ACTION A_Test_Motion:
T_Delay_RB_A_Tool_1 (PT:=T#500MS);
T_Delay_RB_A_Tool_2 (PT:=T#500MS);
IF A_Test_Motion_Run THEN
	CASE Process_A_Test OF
		0: // Point 0
			M_CHOOSE_POS(DATA := Move_Point_Para_A.Hand_Type, ID := 0, XYR_CONST := TRUE, Z_CONST:= FALSE);
			IF NOT Move_Point_Para_A.Enable THEN
				Move_Point_Para_A.Enable := TRUE;
				Move_Point_Para_A.Move_Type := 0;
			END_IF
			IF Move_RB_A.Done AND NOT Move_RB_A.Busy THEN	
				Process_A_Test := Process_A_Test + 5;
				Move_Point_Para_A.Enable := FALSE;
			END_IF;
		5: // Point 1
			M_CHOOSE_POS(DATA := Move_Point_Para_A.Hand_Type, ID := 0, XYR_CONST := FALSE, Z_CONST:= FALSE);
			IF NOT Move_Point_Para_A.Enable THEN
				Move_Point_Para_A.Enable := TRUE;
				Move_Point_Para_A.Move_Type := 0;
			END_IF
			IF Move_RB_A.Done AND NOT Move_RB_A.Busy THEN	
				Process_A_Test := Process_A_Test + 5;
				Move_Point_Para_A.Enable := FALSE;
			END_IF;
		10: // Point 2 - BF Pick T1 - 1
			M_CHOOSE_POS(DATA := Move_Point_Para_A.Hand_Type, ID := 1, XYR_CONST := FALSE, Z_CONST:= FALSE);
			IF NOT Move_Point_Para_A.Enable THEN
				Move_Point_Para_A.Enable := TRUE;
				Move_Point_Para_A.Move_Type := 0;
			END_IF
			IF Move_RB_A.Done AND NOT Move_RB_A.Busy THEN	
				Process_A_Test := Process_A_Test + 10;
				Move_Point_Para_A.Enable := FALSE;
			END_IF;
		20: // Point 3 - Pick Product by Tool 1 - 1
			M_CHOOSE_POS(DATA := Move_Point_Para_A.Hand_Type, ID := 2, XYR_CONST := FALSE, Z_CONST:= FALSE);
			IF NOT Move_Point_Para_A.Enable THEN
				Move_Point_Para_A.Enable := TRUE;
				Move_Point_Para_A.Move_Type := 0;
			END_IF
			IF Move_RB_A.Done AND NOT Move_RB_A.Busy THEN	
				GVL.RB_A_.Tool_1 := 1;
				T_Delay_RB_A_Tool_1.IN := TRUE;
				
			END_IF;
			IF T_Delay_RB_A_Tool_1.Q THEN	
				Move_Point_Para_A.Enable := FALSE;
				T_Delay_RB_A_Tool_1.IN := FALSE;
				Process_A_Test := Process_A_Test + 10;
			END_IF;
		30: // Point 2 - Return BF Pick T1 -1
			M_CHOOSE_POS(DATA := Move_Point_Para_A.Hand_Type, ID := 1, XYR_CONST := FALSE, Z_CONST:= FALSE);
			IF NOT Move_Point_Para_A.Enable THEN
				Move_Point_Para_A.Enable := TRUE;
				Move_Point_Para_A.Move_Type := 0;
			END_IF
			IF Move_RB_A.Done AND NOT Move_RB_A.Busy THEN	
				Process_A_Test := Process_A_Test + 10;
				Move_Point_Para_A.Enable := FALSE;
			END_IF;
				
		40: // Point 4 - BF Place T1 - 1
			M_CHOOSE_POS(DATA := Move_Point_Para_A.Hand_Type, ID := 3, XYR_CONST := FALSE, Z_CONST:= FALSE);
			IF NOT Move_Point_Para_A.Enable THEN
				Move_Point_Para_A.Enable := TRUE;
				Move_Point_Para_A.Move_Type := 0;
			END_IF
			IF Move_RB_A.Done AND NOT Move_RB_A.Busy THEN	
				Process_A_Test := Process_A_Test + 10;
				Move_Point_Para_A.Enable := FALSE;
			END_IF;
		
		50: // Point 5 - Place T1 - 1 
			M_CHOOSE_POS(DATA := Move_Point_Para_A.Hand_Type, ID := 4, XYR_CONST := FALSE, Z_CONST:= FALSE);
			IF NOT Move_Point_Para_A.Enable THEN
				Move_Point_Para_A.Enable := TRUE;
				Move_Point_Para_A.Move_Type := 0;
			END_IF
			IF Move_RB_A.Done AND NOT Move_RB_A.Busy THEN	
				GVL.RB_A_.Tool_1 := 0;
				T_Delay_RB_A_Tool_1.IN := TRUE;
				//Move_Point_Para_A.Enable := FALSE;
			END_IF;
			
			IF T_Delay_RB_A_Tool_1.Q THEN			
				Move_Point_Para_A.Enable := FALSE;
				T_Delay_RB_A_Tool_1.IN := FALSE;
				Process_A_Test := Process_A_Test + 10;
			END_IF
		
		60: // Point 4 - BF Place T1 - 1
			M_CHOOSE_POS(DATA := Move_Point_Para_A.Hand_Type, ID := 3, XYR_CONST := FALSE, Z_CONST:= FALSE);
			IF NOT Move_Point_Para_A.Enable THEN
				Move_Point_Para_A.Enable := TRUE;
				Move_Point_Para_A.Move_Type := 0;
			END_IF
			IF Move_RB_A.Done AND NOT Move_RB_A.Busy THEN	
				Process_A_Test := Process_A_Test + 10;
				Move_Point_Para_A.Enable := FALSE;
			END_IF;
			
		70: // Point 6 - BF Pick T1-2
			M_CHOOSE_POS(DATA := Move_Point_Para_A.Hand_Type, ID := 5, XYR_CONST := FALSE, Z_CONST:= FALSE);
			IF NOT Move_Point_Para_A.Enable THEN
				Move_Point_Para_A.Enable := TRUE;
				Move_Point_Para_A.Move_Type := 0;
			END_IF
			IF Move_RB_A.Done AND NOT Move_RB_A.Busy THEN	
				Process_A_Test := Process_A_Test + 10;
				Move_Point_Para_A.Enable := FALSE;
			END_IF;
		80: // Point 7 - Pick Tool 1 - 2
			M_CHOOSE_POS(DATA := Move_Point_Para_A.Hand_Type, ID := 6, XYR_CONST := FALSE, Z_CONST:= FALSE);
			IF NOT Move_Point_Para_A.Enable THEN
				Move_Point_Para_A.Enable := TRUE;
				Move_Point_Para_A.Move_Type := 0;
			END_IF
			IF Move_RB_A.Done AND NOT Move_RB_A.Busy THEN	
				GVL.RB_A_.Tool_1 := 1;
				T_Delay_RB_A_Tool_2.IN := TRUE;
				//Move_Point_Para_A.Enable := FALSE;
			END_IF;
			IF T_Delay_RB_A_Tool_2.Q THEN
				T_Delay_RB_A_Tool_2.IN := FALSE;
				Move_Point_Para_A.Enable := FALSE;
				Process_A_Test := Process_A_Test + 10;
			END_IF;
		90: // Point 6 - Return BF Pick T1 - 2 
			M_CHOOSE_POS(DATA := Move_Point_Para_A.Hand_Type, ID := 5, XYR_CONST := FALSE, Z_CONST:= FALSE);
			IF NOT Move_Point_Para_A.Enable THEN
				Move_Point_Para_A.Enable := TRUE;
				Move_Point_Para_A.Move_Type := 0;
			END_IF
			IF Move_RB_A.Done AND NOT Move_RB_A.Busy THEN	
				Process_A_Test := Process_A_Test + 10;
				Move_Point_Para_A.Enable := FALSE;
			END_IF;
				
		100: // Point 8 - BF Place T1 - 2 
			M_CHOOSE_POS(DATA := Move_Point_Para_A.Hand_Type, ID := 7, XYR_CONST := FALSE, Z_CONST:= FALSE);
			IF NOT Move_Point_Para_A.Enable THEN
				Move_Point_Para_A.Enable := TRUE;
				Move_Point_Para_A.Move_Type := 0;
			END_IF
			IF Move_RB_A.Done AND NOT Move_RB_A.Busy THEN	
				Process_A_Test := Process_A_Test + 10;
				Move_Point_Para_A.Enable := FALSE;
			END_IF;
		
		110: // Point 9 - Place T2
			M_CHOOSE_POS(DATA := Move_Point_Para_A.Hand_Type, ID := 8, XYR_CONST := FALSE, Z_CONST:= FALSE);
			IF NOT Move_Point_Para_A.Enable THEN
				Move_Point_Para_A.Enable := TRUE;
				Move_Point_Para_A.Move_Type := 0;
			END_IF
			IF Move_RB_A.Done AND NOT Move_RB_A.Busy THEN	
				GVL.RB_A_.Tool_1 := 0;
				T_Delay_RB_A_Tool_2.IN := TRUE;
				//Move_Point_Para_A.Enable := FALSE;
			END_IF;
			
			IF T_Delay_RB_A_Tool_2.Q THEN			
				T_Delay_RB_A_Tool_2.IN := FALSE;
				Move_Point_Para_A.Enable := FALSE;
				Process_A_Test := Process_A_Test + 10;
			END_IF
		
		120: // Point 8 - BF Place T2
			M_CHOOSE_POS(DATA := Move_Point_Para_A.Hand_Type, ID := 7, XYR_CONST := FALSE, Z_CONST:= FALSE);
			IF NOT Move_Point_Para_A.Enable THEN
				Move_Point_Para_A.Enable := TRUE;
				Move_Point_Para_A.Move_Type := 0;
			END_IF
			IF Move_RB_A.Done AND NOT Move_RB_A.Busy THEN	
				Process_A_Test := Process_A_Test + 10;
				Move_Point_Para_A.Enable := FALSE;
			END_IF;
			
		
		130: // WAIT XYR
			Process_A_Test := 5;
			A_Test_Motion_Finish := TRUE;
		
	END_CASE
ELSE
	Process_A_Test := 0;
END_IF
END_ACTION

ACTION B1_Test_Motion:
Ton_Test_B(PT := T#500MS);
T_Delay_RB_B_Tool_1(PT := T#500MS);
T_Delay_RB_B_Tool_2(PT := T#500MS);
IF B_Test_Motion_Run THEN
	CASE Process_B_Test OF
		0: // Point 0
			M_CHOOSE_POS(DATA := Move_Point_Para_B.Hand_Type, ID := 0, XYR_CONST := TRUE, Z_CONST:= FALSE);
			IF NOT Move_Point_Para_B.Enable THEN
				Move_Point_Para_B.Enable := TRUE;
				Move_Point_Para_B.Move_Type := 0;
			END_IF
			IF Move_RB_B.Done AND NOT Move_RB_B.Busy THEN	
				Process_B_Test := Process_B_Test + 5;
				Move_Point_Para_B.Enable := FALSE;
			END_IF;
		5: // Point 1
			M_CHOOSE_POS(DATA := Move_Point_Para_B.Hand_Type, ID := 0, XYR_CONST := FALSE, Z_CONST:= FALSE);
			IF NOT Move_Point_Para_B.Enable THEN
				Move_Point_Para_B.Enable := TRUE;
				Move_Point_Para_B.Move_Type := 0;
			END_IF
			IF Move_RB_B.Done AND NOT Move_RB_B.Busy THEN	
				Process_B_Test := Process_B_Test + 5;
				Move_Point_Para_B.Enable := FALSE;
			END_IF;
		10: // Point 2 - BF Pick T1
			M_CHOOSE_POS(DATA := Move_Point_Para_B.Hand_Type, ID := 1, XYR_CONST := FALSE, Z_CONST:= FALSE);
			IF NOT Move_Point_Para_B.Enable THEN
				Move_Point_Para_B.Enable := TRUE;
				Move_Point_Para_B.Move_Type := 0;
			END_IF
			IF Move_RB_B.Done AND NOT Move_RB_B.Busy THEN	
				Process_B_Test := Process_B_Test + 10;
				Move_Point_Para_B.Enable := FALSE;
			END_IF;
		
		20: // WAIT Timer
			
			Ton_Test_B.IN := TRUE;
			IF Ton_Test_B.Q THEN
				Process_B_Test := 30;
				Ton_Test_B.IN := FALSE;
			END_IF
		30: // Point 3 - Pick T1
			
			M_CHOOSE_POS(DATA := Move_Point_Para_B.Hand_Type, ID := 2, XYR_CONST := FALSE, Z_CONST:= FALSE);
			IF NOT Move_Point_Para_B.Enable THEN
				Move_Point_Para_B.Enable := TRUE;
				Move_Point_Para_B.Move_Type := 0;
			END_IF
			IF Move_RB_B.Done AND NOT Move_RB_B.Busy THEN	
				GVL.RB_B_.Tool_1 := 1;
				T_Delay_RB_B_Tool_1.IN := TRUE;
				
			END_IF;
			IF T_Delay_RB_B_Tool_1.Q THEN
				Move_Point_Para_B.Enable := FALSE;
				T_Delay_RB_B_Tool_1.IN := FALSE;
				Process_B_Test := Process_B_Test + 10;		
			END_IF;
		40: // Point 2 - BF Pick T1
			M_CHOOSE_POS(DATA := Move_Point_Para_B.Hand_Type, ID := 1, XYR_CONST := FALSE, Z_CONST:= FALSE);
			IF NOT Move_Point_Para_B.Enable THEN
				Move_Point_Para_B.Enable := TRUE;
				Move_Point_Para_B.Move_Type := 0;
			END_IF
			IF Move_RB_B.Done AND NOT Move_RB_B.Busy THEN	
				Process_B_Test := Process_B_Test + 10;
				Move_Point_Para_B.Enable := FALSE;
			END_IF;
		50: // Point 4 - BF Place T1
			M_CHOOSE_POS(DATA := Move_Point_Para_B.Hand_Type, ID := 3, XYR_CONST := FALSE, Z_CONST:= FALSE);
			IF NOT Move_Point_Para_B.Enable THEN
				Move_Point_Para_B.Enable := TRUE;
				Move_Point_Para_B.Move_Type := 0;
			END_IF
			IF Move_RB_B.Done AND NOT Move_RB_B.Busy THEN	
				Process_B_Test := Process_B_Test + 10;
				Move_Point_Para_B.Enable := FALSE;
			END_IF;
		
		60: // Point 5 - Place T1
			M_CHOOSE_POS(DATA := Move_Point_Para_B.Hand_Type, ID := 4, XYR_CONST := FALSE, Z_CONST:= FALSE);
			IF NOT Move_Point_Para_B.Enable THEN
				Move_Point_Para_B.Enable := TRUE;
				Move_Point_Para_B.Move_Type := 0;
			END_IF
			IF Move_RB_B.Done AND NOT Move_RB_B.Busy THEN	
				GVL.RB_B_.Tool_1 := 0;
				T_Delay_RB_B_Tool_1.IN := TRUE;
				
			END_IF;
			IF T_Delay_RB_B_Tool_1.Q THEN
				Move_Point_Para_B.Enable := FALSE;
				T_Delay_RB_B_Tool_1.IN := FALSE;
				Process_B_Test := Process_B_Test + 10;
				
			END_IF;
			
		70: // Point 4 - BF Place T1
			M_CHOOSE_POS(DATA := Move_Point_Para_B.Hand_Type, ID := 3, XYR_CONST := FALSE, Z_CONST:= FALSE);
			IF NOT Move_Point_Para_B.Enable THEN
				Move_Point_Para_B.Enable := TRUE;
				Move_Point_Para_B.Move_Type := 0;
			END_IF
			IF Move_RB_B.Done AND NOT Move_RB_B.Busy THEN	
				Process_B_Test := Process_B_Test + 10;
				Move_Point_Para_B.Enable := FALSE;
			END_IF;
			
		80: // Point 6 - BF Pick T2
			M_CHOOSE_POS(DATA := Move_Point_Para_B.Hand_Type, ID := 5, XYR_CONST := FALSE, Z_CONST:= FALSE);
			IF NOT Move_Point_Para_B.Enable THEN
				Move_Point_Para_B.Enable := TRUE;
				Move_Point_Para_B.Move_Type := 0;
			END_IF
			IF Move_RB_B.Done AND NOT Move_RB_B.Busy THEN	
				Process_B_Test := Process_B_Test + 10;
				Move_Point_Para_B.Enable := FALSE;
			END_IF;
		

		90: // Point 7 - Pick T2
			M_CHOOSE_POS(DATA := Move_Point_Para_B.Hand_Type, ID := 6, XYR_CONST := FALSE, Z_CONST:= FALSE);
			IF NOT Move_Point_Para_B.Enable THEN
				Move_Point_Para_B.Enable := TRUE;
				Move_Point_Para_B.Move_Type := 0;
			END_IF
			IF Move_RB_B.Done AND NOT Move_RB_B.Busy THEN	
				GVL.RB_B_.Tool_1 := 1;
				T_Delay_RB_B_Tool_2.IN := TRUE;
				
			END_IF;
			IF T_Delay_RB_B_Tool_2.Q THEN
				Move_Point_Para_B.Enable := FALSE;
				T_Delay_RB_B_Tool_2.IN := FALSE;
				Process_B_Test := Process_B_Test + 10;
				
			END_IF;
		100: // Point 6 - BF Pick T2
			M_CHOOSE_POS(DATA := Move_Point_Para_B.Hand_Type, ID := 5, XYR_CONST := FALSE, Z_CONST:= FALSE);
			IF NOT Move_Point_Para_B.Enable THEN
				Move_Point_Para_B.Enable := TRUE;
				Move_Point_Para_B.Move_Type := 0;
			END_IF
			IF Move_RB_B.Done AND NOT Move_RB_B.Busy THEN	
				Process_B_Test := Process_B_Test + 10;
				Move_Point_Para_B.Enable := FALSE;
			END_IF;
		110: // Point 8 - BF Place T2
			M_CHOOSE_POS(DATA := Move_Point_Para_B.Hand_Type, ID := 7, XYR_CONST := FALSE, Z_CONST:= FALSE);
			IF NOT Move_Point_Para_B.Enable THEN
				Move_Point_Para_B.Enable := TRUE;
				Move_Point_Para_B.Move_Type := 0;
			END_IF
			IF Move_RB_B.Done AND NOT Move_RB_B.Busy THEN	
				Process_B_Test := Process_B_Test + 10;
				Move_Point_Para_B.Enable := FALSE;
			END_IF;
		
		120: // Point 9 - Place T2
			M_CHOOSE_POS(DATA := Move_Point_Para_B.Hand_Type, ID := 8, XYR_CONST := FALSE, Z_CONST:= FALSE);
			IF NOT Move_Point_Para_B.Enable THEN
				Move_Point_Para_B.Enable := TRUE;
				Move_Point_Para_B.Move_Type := 0;
			END_IF
			IF Move_RB_B.Done AND NOT Move_RB_B.Busy THEN	
				GVL.RB_B_.Tool_1 := 0;
				T_Delay_RB_B_Tool_2.IN := TRUE;
				
			END_IF;
			IF T_Delay_RB_B_Tool_2.Q THEN
				Move_Point_Para_B.Enable := FALSE;
				T_Delay_RB_B_Tool_2.IN := FALSE;
				Process_B_Test := Process_B_Test + 10;
				
			END_IF;
			
		130: // Point 8 - BF Place T2
			M_CHOOSE_POS(DATA := Move_Point_Para_B.Hand_Type, ID := 7, XYR_CONST := FALSE, Z_CONST:= FALSE);
			IF NOT Move_Point_Para_B.Enable THEN
				Move_Point_Para_B.Enable := TRUE;
				Move_Point_Para_B.Move_Type := 0;
			END_IF
			IF Move_RB_B.Done AND NOT Move_RB_B.Busy THEN	
				Process_B_Test := Process_B_Test + 10;
				Move_Point_Para_B.Enable := FALSE;
			END_IF;
			
			
		140: // Finish
			//Ton_Test_B.IN := FALSE;
			Process_B_Test := 5;
			A_Test_Motion_Finish := TRUE;
			
		
	END_CASE
ELSE
	Process_B_Test := 0;
END_IF
END_ACTION

ACTION _Main_Process_Test_VS:
// PROCESS 
IF Ena_Test THEN
	GVL.RB_A.COORD := 1;
	GVL.RB_B.COORD := 1;
	IF NOT Just_Start_Test THEN
		A_Test_Motion_Run := FALSE;
		B_Test_Motion_Run := FALSE;
		Process_B_Test := 0;
		Process_A_Test := 0;
	END_IF
	Just_Start_Test := TRUE;
	A_Test_Motion_Run := TRUE;
	A_Test_Motion_VS();
// 	B_Test_Motion_Run := TRUE;
// 	B1_Test_Motion_VS();

ELSIF NOT Ena_Test THEN

	A_Test_Motion_Run := FALSE;
	B_Test_Motion_Run := FALSE;
	Process_B_Test := 0;
	Process_A_Test := 0;
	
END_IF	 
{endregion}
END_ACTION

ACTION A_Test_Motion_VS:
Ton_Test_A(PT := T#500MS);
IF A_Test_Motion_Run THEN
	CASE Process_A_Test OF
		0: // Point 1 - Wait
			M_CHOOSE_POS(DATA := Move_Point_Para_A.Hand_Type, ID := 0, XYR_CONST := FALSE, Z_CONST:= FALSE);
			IF NOT Move_Point_Para_A.Enable THEN
				Move_Point_Para_A.Enable := TRUE;
				Move_Point_Para_A.Move_Type := 0;
			END_IF
			IF Move_RB_A.Done AND NOT Move_RB_A.Busy THEN	
				Process_A_Test := Process_A_Test + 10;
				Move_Point_Para_A.Enable := FALSE;
			END_IF;
		10: // Point 2 - BF Pick T1
			M_CHOOSE_POS(DATA := Move_Point_Para_A.Hand_Type, ID := 1, XYR_CONST := FALSE, Z_CONST:= FALSE);
			IF NOT Move_Point_Para_A.Enable THEN
				Move_Point_Para_A.Enable := TRUE;
				Move_Point_Para_A.Move_Type := 0;
			END_IF
			IF Move_RB_A.Done AND NOT Move_RB_A.Busy THEN	
				Process_A_Test := Process_A_Test + 10;
				Move_Point_Para_A.Enable := FALSE;
			END_IF;
		20: // Point 3 - Pick T1
			M_CHOOSE_POS(DATA := Move_Point_Para_A.Hand_Type, ID := 2, XYR_CONST := FALSE, Z_CONST:= FALSE);
			IF NOT Move_Point_Para_A.Enable THEN
				Move_Point_Para_A.Enable := TRUE;
				Move_Point_Para_A.Move_Type := 0;
			END_IF
			IF Move_RB_A.Done AND NOT Move_RB_A.Busy THEN	
				Process_A_Test := Process_A_Test + 10;
				Move_Point_Para_A.Enable := FALSE;
			END_IF;
		30: // Point 4 - BF Pick T1
			M_CHOOSE_POS(DATA := Move_Point_Para_A.Hand_Type, ID := 3, XYR_CONST := FALSE, Z_CONST:= FALSE);
			IF NOT Move_Point_Para_A.Enable THEN
				Move_Point_Para_A.Enable := TRUE;
				Move_Point_Para_A.Move_Type := 0;
			END_IF
			IF Move_RB_A.Done AND NOT Move_RB_A.Busy THEN	
				Process_A_Test := Process_A_Test + 10;
				Move_Point_Para_A.Enable := FALSE;
			END_IF;
				
		40: // Point 5 - Trigger VS
			M_CHOOSE_POS(DATA := Move_Point_Para_A.Hand_Type, ID := 4, XYR_CONST := FALSE, Z_CONST:= FALSE);
			IF NOT Move_Point_Para_A.Enable THEN
				Move_Point_Para_A.Enable := TRUE;
				Move_Point_Para_A.Move_Type := 0;
			END_IF
			IF Move_RB_A.Done AND NOT Move_RB_A.Busy THEN	
				Process_A_Test := Process_A_Test + 10;
				Move_Point_Para_A.Enable := FALSE;
			END_IF;
			
		50: // WAIT Timer
			
			Ton_Test_A.IN := TRUE;
			IF Ton_Test_A.Q THEN
				Process_A_Test := Process_A_Test + 10;
				Ton_Test_A.IN := FALSE;
			END_IF
			
		60: // Trigger VS
			
			IF ( NOT GVL.Data_Calib_RB[0].Run_No_Trigger) THEN
				GVL.Auto_VS_RB[0].Enable_FB_Trigger_VS := TRUE;
				GVL.Auto_VS_RB[0].Start_FB_Trigger_VS := TRUE;
			END_IF
			
			IF ((Trigger_VS_FB[0].DoneAll AND NOT Trigger_VS_FB[0].Busy) OR GVL.Data_Calib_RB[0].Run_No_Trigger ) THEN
				GVL.Auto_VS_RB[0].Enable_FB_Trigger_VS := FALSE;
				GVL.Auto_VS_RB[0].Start_FB_Trigger_VS := FALSE;
				Process_A_Test := Process_A_Test + 10;
			END_IF;	
			
		70: // WAIT XYR
			Process_A_Test := 0;
			A_Test_Motion_Finish := TRUE;
		
	END_CASE
ELSE
	Process_A_Test := 0;
END_IF
END_ACTION

ACTION B1_Test_Motion_VS:
Ton_Test_B(PT := T#500MS);
IF B_Test_Motion_Run THEN
	CASE Process_B_Test OF
		0: // Point 1 - Wait
			M_CHOOSE_POS(DATA := Move_Point_Para_B.Hand_Type, ID := 0, XYR_CONST := FALSE, Z_CONST:= FALSE);
			IF NOT Move_Point_Para_B.Enable THEN
				Move_Point_Para_B.Enable := TRUE;
				Move_Point_Para_B.Move_Type := 0;
			END_IF
			IF Move_RB_B.Done AND NOT Move_RB_B.Busy THEN	
				Process_B_Test := Process_B_Test + 10;
				Move_Point_Para_B.Enable := FALSE;
			END_IF;
		10: // Point 2 - BF Pick T1
			M_CHOOSE_POS(DATA := Move_Point_Para_B.Hand_Type, ID := 1, XYR_CONST := FALSE, Z_CONST:= FALSE);
			IF NOT Move_Point_Para_B.Enable THEN
				Move_Point_Para_B.Enable := TRUE;
				Move_Point_Para_B.Move_Type := 0;
			END_IF
			IF Move_RB_B.Done AND NOT Move_RB_B.Busy THEN	
				Process_B_Test := Process_B_Test + 10;
				Move_Point_Para_B.Enable := FALSE;
			END_IF;
		
		20: // WAIT Timer
			Process_B_Test := Process_B_Test + 10;
// 			Ton_Test_B.IN := TRUE;
// 			IF Ton_Test_B.Q THEN
// 				Process_B_Test := 30;
// 				Ton_Test_B.IN := FALSE;
// 			END_IF
		30: // Point 3 - Pick T1
			
			M_CHOOSE_POS(DATA := Move_Point_Para_B.Hand_Type, ID := 2, XYR_CONST := FALSE, Z_CONST:= FALSE);
			IF NOT Move_Point_Para_B.Enable THEN
				Move_Point_Para_B.Enable := TRUE;
				Move_Point_Para_B.Move_Type := 0;
			END_IF
			IF Move_RB_B.Done AND NOT Move_RB_B.Busy THEN	
				Process_B_Test := Process_B_Test + 10;
				Move_Point_Para_B.Enable := FALSE;
			END_IF;
		
		40: // Point 4 - BF Pick T1
			M_CHOOSE_POS(DATA := Move_Point_Para_B.Hand_Type, ID := 3, XYR_CONST := FALSE, Z_CONST:= FALSE);
			IF NOT Move_Point_Para_B.Enable THEN
				Move_Point_Para_B.Enable := TRUE;
				Move_Point_Para_B.Move_Type := 0;
			END_IF
			IF Move_RB_B.Done AND NOT Move_RB_B.Busy THEN	
				Process_B_Test := Process_B_Test + 10;
				Move_Point_Para_B.Enable := FALSE;
			END_IF;
		50: // Point 5 - Trigger VS
			M_CHOOSE_POS(DATA := Move_Point_Para_B.Hand_Type, ID := 4, XYR_CONST := FALSE, Z_CONST:= FALSE);
			IF NOT Move_Point_Para_B.Enable THEN
				Move_Point_Para_B.Enable := TRUE;
				Move_Point_Para_B.Move_Type := 0;
			END_IF
			IF Move_RB_B.Done AND NOT Move_RB_B.Busy THEN	
				Process_B_Test := Process_B_Test + 10;
				Move_Point_Para_B.Enable := FALSE;
			END_IF;
		60: // WAIT Timer
			
			Ton_Test_B.IN := TRUE;
			IF Ton_Test_B.Q THEN
				Process_B_Test := Process_B_Test + 10;
				Ton_Test_B.IN := FALSE;
			END_IF
			
		70: // Trigger VS
			IF ( NOT GVL.Data_Calib_RB[0].Run_No_Trigger) THEN
				GVL.Auto_VS_RB[0].Enable_FB_Trigger_VS := TRUE;
				GVL.Auto_VS_RB[0].Start_FB_Trigger_VS := TRUE;
			END_IF
			
			IF ((Trigger_VS_FB[0].DoneAll AND NOT Trigger_VS_FB[0].Busy) OR GVL.Data_Calib_RB[0].Run_No_Trigger ) THEN
				GVL.Auto_VS_RB[0].Enable_FB_Trigger_VS := FALSE;
				GVL.Auto_VS_RB[0].Start_FB_Trigger_VS := FALSE;
				Process_B_Test := Process_B_Test + 10;
			END_IF;
	
		80: // Finish
			//Ton_Test_B.IN := FALSE;
			Process_B_Test := 0;
			A_Test_Motion_Finish := TRUE;
			
		
	END_CASE
ELSE
	Process_B_Test := 0;
END_IF
END_ACTION

ACTION _Main_Process_4:
// Check Pos cmp

B_Allow_NextStep := NOT GVL_2.Process3.Auto_Man_B OR nextstepRtrigB.Q;
nextstepRtrigB(CLK := ( GVL_2.Process3.Auto_Man_B AND GVL_2.Process3.NextStep_B));
A_Allow_NextStep := NOT GVL_2.Process3.Auto_Man_A OR nextstepRtrigA.Q;
nextstepRtrigA(CLK := ( GVL_2.Process3.Auto_Man_A AND GVL_2.Process3.NextStep_A));
// Clear Data
IF NOT GVL.Pro4_.Process.Clear_Data THEN
	// ko làm gì
ELSE
	GVL.Pro4_.Process.DATA_MC_TS := 0;
	GVL.Pro4_.Process.DATA_MC_VS := 0;
	GVL.Pro4_.Process.DATA_TOOL_A1_IN := 0;
	GVL.Pro4_.Process.DATA_TOOL_A2_OUT := 0;
	GVL.Pro4_.Process.DATA_TOOL_B1_IN := 0;
	GVL.Pro4_.Process.DATA_TOOL_A1_IN_OLD := 0;	
END_IF



// PROCESS 
IF Ena4 THEN
// cv-ng
CNV_NG();	
// Process MC1
Pro_MC1_4_();
// Process MC2
Pro_MC2_4_();	
// trigger
B_Trigger_4();
////// process robot A
A0_Wait_4();
A1_Pick_T1_4();
A2_Place_T1_OK_4();
A3_Place_T1_NG_4();
A4_Pick_T2_4();
A5_Place_T2_OK_4();
A6_Place_T2_NG_4();
A7_Barcode_T1_4();
A8_Place_T2_NG_TS_4();
	CASE Pro_A4 OF
	0: // INIT
			
			GVL.RB_A.COORD := 1;
			RBA_BufferMode := 0; 
	 		Wait_A4_Finish			:= FALSE;
			Pick_A4_T1_Finish 		:= FALSE;
			Pick_A4_T2_Finish		:= FALSE;
			Barcode_A4_Finish		:= FALSE;
			Place_OK_A4_T1_Finish 	:= FALSE;
			Place_Ok_A4_T2_Finish 	:= FALSE;
			Place_NG_A4_T1_Finish 	:= FALSE;
			Place_NG_A4_T2_Finish 	:= FALSE;
			Place_NG_TS_A4_T2_Finish	:= FALSE;
			
	 		Wait_A4_Run				:= FALSE;
			Pick_A4_T1_Run			:= FALSE;
			Pick_A4_T2_Run			:= FALSE;
			Barcode_A4_Run			:= FALSE;
			Place_OK_A4_T1_Run	 	:= FALSE;
			Place_Ok_A4_T2_Run	 	:= FALSE;
			Place_NG_A4_T1_Run	 	:= FALSE;
			Place_NG_A4_T2_Run		:= FALSE;			
			Place_NG_TS_A4_T2_Run	:= FALSE;	
			Pro_A4_BF := 0; // namnv
			Pro_A4 := Pro_A4 + 10; 
			
	10: // CALL WAIT	
		LOG_A.Write('Robot A to Wait');	
		IF NOT Wait_A4_Run THEN
			RBA_BufferMode := 0;
			Wait_A4_Run := TRUE;
		END_IF
		IF Wait_A4_Finish AND A_Allow_NextStep THEN
			Wait_A4_Run := FALSE;
			Pro_A4_BF := 10; // namnv
			Pro_A4 := Pro_A4 + 10;
		END_IF;		
	20: // CHECK PICK OR PLACE T1
			
		 	Wait_A4_Finish			:= FALSE;
			Pick_A4_T1_Finish 		:= FALSE;
			Pick_A4_T2_Finish		:= FALSE;
			Barcode_A4_Finish		:= FALSE;
			Place_OK_A4_T1_Finish 	:= FALSE;
			Place_Ok_A4_T2_Finish 	:= FALSE;
			Place_NG_A4_T1_Finish 	:= FALSE;
			Place_NG_A4_T2_Finish 	:= FALSE;
			Place_NG_TS_A4_T2_Finish 	:= FALSE;
			
			CASE GVL.Pro4_.Process.DATA_TOOL_A1_IN OF
				0: // none
					Pro_A4 := 30; // Pick T1
				1: // Barcode
					Pro_A4 := 40; // Barcode T1
				2: // Ok
					CASE GVL.Pro4_.Process.DATA_MC_VS OF
						2: 
							Pro_A4 := 50; // Place T1 OK => MC2
						3: 
							Pro_A4 := 25; // CHECK PICK OR PLACE T2
						4: 
							Pro_A4 := 25;
						5: 
							Pro_A4 := 25;
					END_CASE;
					
				3: // NG
					// Pro_A4 := 60;	
					// namnv NG cung van dat vao may Vision
					CASE GVL.Pro4_.Process.DATA_MC_VS OF
						2: 
							Pro_A4 := 50; // Place T1 NG => MC2
						3: 
							Pro_A4 := 25; // CHECK PICK OR PLACE T2
						4: 
							Pro_A4 := 25;
							//namnv
						5: 
							Pro_A4 := 25;	
							
					END_CASE;
					
			END_CASE
			// Pro_A4_BF := 20; // namnv
	25: // CHECK PICK OR PLACE T2
			CASE GVL.Pro4_.Process.DATA_TOOL_A2_OUT OF
				0: // none
					Pro_A4 := 70; // pick T2
				1: // have
					//Pro_B3 := 80; // Place OK CNV
				2: // OK
					Pro_A4 := 80; // Place OK CNV
				3: // NG - VS
					Pro_A4 := 90; // Place NG-VS CNV
				// namnv
				4: // NG - TS
					Pro_A4 := 100; // Place NG-TS CNV
			END_CASE	
			// Pro_A4_BF := 25; // namnv	
	30: // Pick T1
		 //DATA_MC1 := 3;
		 LOG_A.Write('Robot A Pick T1');
// 		IF NOT Pick_A4_T1_Run  AND (GVL.Pro4_.Process.DATA_MC_TS = 3 OR GVL.Pro4_.Process.DATA_MC_TS = 4) THEN
		//IF NOT Pick_B3_T1_Run THEN	
		// namnv0204
		IF NOT Pick_A4_T1_Run  AND (GVL.Pro4_.Process.DATA_MC_TS = 3 OR GVL.Pro4_.Process.DATA_MC_TS = 4 OR GVL.Pro4_.Process.DATA_MC_TS = 1) THEN
			RBA_BufferMode := 0;
			Pick_A4_T1_Run := TRUE;
		ELSIF NOT Pick_A4_T1_Run AND GVL.Pro4_.Process.DATA_MC_TS <> 3 AND GVL.Pro4_.Process.DATA_MC_TS <> 4 AND GVL.Pro4_.Process.DATA_MC_TS <> 1 THEN
			Pro_A4 := 25;
			Pro_A4_BF := 30; // namnv
		END_IF
		IF Pick_A4_T1_Finish AND A_Allow_NextStep THEN
			Pick_A4_T1_Run := FALSE;
			// Pro_A4 := 40;
			// namnv - khong cho di ra barcode luon
			Pro_A4 := 20;
			Pro_A4_BF := 30; // namnv
		END_IF;
		
	40: // Barcode T1
		LOG_A.Write('Robot A barcode T1');
		IF NOT Barcode_A4_Run THEN
			RBA_BufferMode := 0;
			Barcode_A4_Run := TRUE;
		END_IF
		IF Barcode_A4_Finish AND A_Allow_NextStep THEN
			Barcode_A4_Run := FALSE;
			// Pro_A4 := 10;
			Pro_A4 := 20;  // Khong cho chay ve wait nua  Namnv
			Pro_A4_BF := 40; // namnv
		END_IF;		
		
	50: // Place T1 OK/NG => MC2
		//DATA_MC2 := 2;
		LOG_A.Write('Robot A Place T1 OK');
		RBA_BufferMode := 1;
		IF NOT Place_OK_A4_T1_Run AND GVL.Pro4_.Process.DATA_MC_VS = 2 THEN
	
			Place_OK_A4_T1_Run := TRUE;
		END_IF
		IF Place_OK_A4_T1_Finish AND A_Allow_NextStep THEN
			Place_OK_A4_T1_Run := FALSE;
			Pro_A4 := 25;
			Pro_A4_BF := 50; // namnv
		END_IF;	
		
	60: // Place T1 NG => CNV TS NG
// 		IF NOT Place_NG_A4_T1_Run  THEN
// 			RBA_BufferMode := 1;
// 			Place_NG_A4_T1_Run := TRUE;
// 		END_IF
// 		IF Place_NG_A4_T1_Finish AND A_Allow_NextStep THEN
// 			Place_NG_A4_T1_Run := FALSE;
// 			Pro_A4 := 10;
// 			Pro_A4_BF := 60; // namnv
// 		END_IF;			
		
				
		
	70: // PICK T2
		//DATA_MC2 := 3;
		//IF NOT Pick_A4_T2_Run  AND ( GVL.Pro4_.Process.DATA_MC_VS = 3 OR GVL.Pro4_.Process.DATA_MC_VS = 4 ) THEN
		LOG_A.Write('Robot A Pick T2');
		IF NOT Pick_A4_T2_Run  AND ( GVL.Pro4_.Process.DATA_MC_VS = 3 OR GVL.Pro4_.Process.DATA_MC_VS = 4 OR GVL.Pro4_.Process.DATA_MC_VS = 5 ) THEN
			RBA_BufferMode := 1;
			Pick_A4_T2_Run := TRUE;
		ELSIF NOT Pick_A4_T2_Run AND( GVL.Pro4_.Process.DATA_MC_VS = 1 OR GVL.Pro4_.Process.DATA_MC_VS = 2) AND ( GVL.Pro4_.Process.DATA_MC_TS = 1 OR GVL.Pro4_.Process.DATA_MC_TS = 3 OR GVL.Pro4_.Process.DATA_MC_TS = 4 ) THEN
			Pro_A4 := 10;
			Pro_A4_BF := 70; // namnv
		END_IF
		IF Pick_A4_T2_Finish AND A_Allow_NextStep THEN
			Pick_A4_T2_Run := FALSE;
			Pro_A4 := 20;
			Pro_A4_BF := 70; // namnv
		END_IF;	
		
	 80: // PLACE T2 OK => CNV OK
		 LOG_A.Write('Robot A Place T2 OK');
		IF NOT Place_Ok_A4_T2_Run   THEN
			Place_Ok_A4_T2_Run := TRUE;
		END_IF
		IF Place_Ok_A4_T2_Finish AND A_Allow_NextStep THEN
			Place_Ok_A4_T2_Run := FALSE;
			Pro_A4 := 10;
			Pro_A4_BF := 80; // namnv
			//GVL.Pro4_.Auto.Nb_Pro_OK := GVL.Pro4_.Auto.Nb_Pro_OK + 1; 
			// namnv1104
			Nb_NG_TS_Cur := 0;
			Nb_NG_VS_Cur := 0;
		END_IF;		 
		
	 90: // PLACE T2 NG => CNV NG VS
		 LOG_A.Write('Robot A Place T2 NG');
		IF NOT Place_NG_A4_T2_Run  THEN
			Place_NG_A4_T2_Run := TRUE;
		END_IF
		IF Place_NG_A4_T2_Finish AND A_Allow_NextStep THEN
			Place_NG_A4_T2_Run := FALSE;
// 			Pro_A4 := 10;
// 			Pro_A4_BF := 90; // namnv
			//GVL.Pro4_.Auto.Nb_Pro_NG := GVL.Pro4_.Auto.Nb_Pro_NG + 1;
			// namnv1104
			IF Nb_NG_VS_Cur < GVL.Pro4_.Auto.Nb_NG_VS_Limit THEN
				Nb_NG_VS_Cur := Nb_NG_VS_Cur + 1;
			END_IF
				
			IF (Nb_NG_VS_Cur >= GVL.Pro4_.Auto.Nb_NG_VS_Limit) THEN
				GVL.Alarm_P4.Alarm_Limit_NG_VS := TRUE;
			ELSE
				GVL.Alarm_P4.Alarm_Limit_NG_VS := FALSE;
			END_IF
			IF (Nb_NG_VS_Cur < GVL.Pro4_.Auto.Nb_NG_VS_Limit) OR GVL.ConfirmNG_VS THEN
				Pro_A4 := 10;
				Pro_A4_BF := 90; // namnv
				IF GVL.ConfirmNG_VS THEN
					Nb_NG_VS_Cur := 0;
					GVL.Alarm_P4.Alarm_Limit_NG_VS := FALSE;
				END_IF
				GVL.ConfirmNG_VS := FALSE;
			END_IF
		END_IF;		
	
	// namnv - them chu trinh tha hang NG Test song tu may VS	
	 100:
	 	LOG_A.Write('Robot A Place T1 TS NG');
		IF NOT Place_NG_TS_A4_T2_Run  THEN
			Place_NG_TS_A4_T2_Run := TRUE;
		END_IF
		IF Place_NG_TS_A4_T2_Finish AND A_Allow_NextStep THEN
			Place_NG_TS_A4_T2_Run := FALSE;
// 			Pro_A4 := 10;
// 			Pro_A4_BF := 100; // namnv
			
			// GVL.Pro4_.Auto.Nb_Pro_NG := GVL.Pro4_.Auto.Nb_Pro_NG + 1;
			// namnv1104
			IF Nb_NG_TS_Cur < GVL.Pro4_.Auto.Nb_NG_TS_Limit THEN
				Nb_NG_TS_Cur := Nb_NG_TS_Cur + 1;
			END_IF
			IF (Nb_NG_TS_Cur >= GVL.Pro4_.Auto.Nb_NG_TS_Limit) THEN
				GVL.Alarm_P4.Alarm_Limit_NG_TS := TRUE;
			ELSE
				GVL.Alarm_P4.Alarm_Limit_NG_TS := FALSE;
			END_IF
			IF (Nb_NG_TS_Cur < GVL.Pro4_.Auto.Nb_NG_TS_Limit) OR GVL.ConfirmNG_TS THEN
				Pro_A4 := 10;
				Pro_A4_BF := 100; // namnv
				IF GVL.ConfirmNG_TS THEN
					Nb_NG_TS_Cur := 0;
					GVL.Alarm_P4.Alarm_Limit_NG_TS := FALSE;
				END_IF
				GVL.ConfirmNG_VS := FALSE;
				
			END_IF
		END_IF;
 	
		
	END_CASE
///////////////////////////////////////////////////////////////////////////////// RB A	
B0_wait_4();
B1_Pick_T1_4();
B2_PLace_T1_4();
B3_Barcode_4();
IF PRO_B4_[1] = 30 OR PRO_B4_[2] = 60 OR PRO_B4_[3] = 30 THEN  Project_4_Delay_B(IN:= TRUE, PT := T#1S); END_IF;

  CASE Pro_B4 OF
	0: // INIT
			
			GVL.RB_B.COORD := 1;
			// GVL.Pro4_.ST_MC.Mode_Dry := FALSE;
	 		Wait_B4_Finish		:= FALSE;
			Pick_B4_Finish 		:= FALSE;
			Barcode_B4_Finish 	:= FALSE;
			Place_B4_Finish		:= FALSE;
			Trigger_B4_Finish	:= FALSE;
			Wait_B4_Run			:= FALSE;
			Pick_B4_Run			:= FALSE;
			Barcode_B4_Run 		:= FALSE;
			Place_B4_Run		:= FALSE;
			Trigger_B4_Run		:= FALSE;
			GVL.Pro4_.Auto.comfirm_Reduct_Pro := FALSE;
			GVL.Pro4_.Auto.Alarm_Not_barcode := FALSE;
			Pro_B4 := Pro_B4 + 10; 
		
	10: // CALL WAIT	
		LOG_B.Write('Robot B to Wait');		
		IF NOT Wait_B4_Run THEN
			Wait_B4_Run := TRUE;
		END_IF
		IF Wait_B4_Finish AND B_Allow_NextStep THEN
			Wait_B4_Run := FALSE;
			Pro_B4 := Pro_B4 + 10;
		END_IF;		
	20: // CHECK PICK OR PLACE
			Wait_B4_Finish		:= FALSE;
			Pick_B4_Finish 		:= FALSE;
			Barcode_B4_Finish 	:= FALSE;
			Place_B4_Finish		:= FALSE;
		CASE GVL.Pro4_.Process.DATA_TOOL_B1_IN OF
			0: // none
				Pro_B4 := 30;
			1: // Have - Trigger Vision
				IF NOT GVL.Pro4_.ST_MC.Mode_Skip_VS_Align THEN
					Pro_B4  := 35;
				ELSE
					Pro_B4 := 40;
				END_IF;
			2: // Barcode Done To Place
				Pro_B4  := 50;
			3: // Trigger Done - To Barcode
				Pro_B4 := 40;
		END_CASE
	30: // Pick 
		LOG_B.Write('Robot B Pick T1');
// 		IF GVL.Pro4_.Signal_In.T_Cv_In_1.q = TRUE OR GVL.Pro4_.ST_MC.Mode_Dry THEN
// 			GVL.Pro4_.Auto.Lighting_On_Off := TRUE;
// 			on_Cam(IN := TRUE, PT := T#500MS, Q =>, ET =>);
// 			IF on_Cam.Q THEN
// 				GVL_2.Process3.Trigger := TRUE;
// 				ALLOW_PICK_CNV := TRUE;
// 			END_IF
// 		ELSE
// 			GVL_2.Process3.Trigger := FALSE;
// 			ALLOW_PICK_CNV := FALSE;
// 			GVL.Pro4_.Auto.Lighting_On_Off := FALSE;
// 		END_IF;
		IF GVL.Pro4_.Signal_In.T_Cv_In_1.q = TRUE OR GVL.Pro4_.ST_MC.Mode_Dry THEN
			ALLOW_PICK_CNV := TRUE;
		ELSE
			ALLOW_PICK_CNV := FALSE;
		END_IF;
		IF (NOT GVL.Pro4_.ST_MC.Mode_Skip_VS_Align) THEN
			GVL.Pro4_.Auto.Lighting_On_Off := TRUE;
		END_IF;
		IF NOT Pick_B4_Run  AND ALLOW_PICK_CNV THEN
			on_Cam.IN := FALSE;
			Pick_B4_Run := TRUE;
		END_IF
		IF Pick_B4_Finish AND B_Allow_NextStep THEN
			Pick_B4_Run := FALSE;
			Pro_B4 := 20;
			
		END_IF;
	35: // Trigger vision
		LOG_B.Write('Robot B Trigger Vision T1');
		IF NOT Trigger_B4_Run THEN
			Trigger_B4_Run := TRUE;
		END_IF
		IF Trigger_B4_Finish AND B_Allow_NextStep THEN
			Trigger_B4_Run := FALSE;

			Pro_B4 := 20; /// ok Trigger >> Doc Barcode
			GVL.Pro4_.Auto.Lighting_On_Off := FALSE;
		END_IF;	
	40: // Barcode
		LOG_B.Write('Robot B Barcode T1');
		IF NOT Barcode_B4_Run THEN
			Barcode_B4_Run := TRUE;
		END_IF
		IF Barcode_B4_Finish AND B_Allow_NextStep THEN
			Barcode_B4_Run := FALSE;
			GVL.Pro4_.Auto.comfirm_Reduct_Pro := FALSE;
			GVL.Pro4_.Auto.Alarm_Not_barcode := FALSE;
			Pro_B4 := 20; /// ok barcode >> place Ts
		END_IF;		
	50: // Place
		LOG_B.Write('Robot B PLace T1');
		//DATA_MC1 := 2;
		// IF NOT Place_B4_Run AND GVL.Pro4_.Process.DATA_MC_TS = 2 THEN
		IF NOT Place_B4_Run AND (GVL.Pro4_.Process.DATA_MC_TS = 2 OR GVL.Pro4_.Process.DATA_MC_TS = 1) THEN
			Place_B4_Run := TRUE;	
		END_IF
		IF Place_B4_Finish AND B_Allow_NextStep THEN
			Place_B4_Run := FALSE;
			Pro_B4 := 0;
		END_IF;		
   END_CASE

ELSIF NOT Ena4 THEN

	
	GVL.Pro4_.Auto.centering_ts_On_Off  := FALSE;
	GVL.Pro4_.Auto.Lighting_On_Off := FALSE;
	D_Barcode_Ts := 0;
	D_Barcode_vs := 0;
	Pro_B4 		:= 0;
	Pro_A4		:= 0;
	Pro_MC1_4	:= 0;
	Pro_MC2_4	:= 0;
	B4_Run_L 	:= FALSE;	
	B4_Run_P 	:= FALSE;
	A4_Run_L	:= FALSE;
	A4_Run_P 	:= FALSE;
	PRO_B4_ [0] := 0;
	PRO_B4_ [1] := 0;
	PRO_B4_ [2] := 0;
	PRO_B4_ [3] := 0;
	PRO_B4_ [4] := 0;
	PRO_B4_ [5] := 0;
	PRO_B4_ [6] := 0;
	PRO_B4_ [7] := 0;
	PRO_B4_ [8] := 0;
	PRO_B4_ [9] := 0;
	
	PRO_A4_ [0] := 0;
	PRO_A4_ [1] := 0;
	PRO_A4_ [2] := 0;
	PRO_A4_ [3] := 0;
	PRO_A4_ [4] := 0;
	PRO_A4_ [5] := 0;
	PRO_A4_ [6] := 0;
	PRO_A4_ [7] := 0;
	PRO_A4_ [8] := 0;
	PRO_A4_ [9] := 0;
	
END_IF	 
{endregion}
END_ACTION

ACTION A0_Wait_4:
// về wait robot B (teaching Point 1)
IF Wait_A4_Run THEN
	CASE PRO_A4_[0] OF
		0: // RESET
				A4_Run_L	 := FALSE;
				A4_Run_P	 := FALSE;
				A_Comp		 := FALSE;			
				PRO_A4_[0] := PRO_A4_[0] + 10;
		10: // Z WAIT
			M_CHOOSE_POS(DATA := 0, ID := 0, XYR_CONST := TRUE, Z_CONST:= FALSE);
			IF NOT A4_Run_P THEN
				A_Comp := FALSE;
				A4_Run_P := TRUE;
			END_IF		
			IF MOVP_A.Error OR MOVL_A.Error THEN
				A4_Run_L	:= FALSE;
				A4_Run_P 	:= FALSE;	 
			END_IF;				
			IF A_Comp AND A4_Run_P AND A_Allow_NextStep THEN
				A4_Run_L	 := FALSE;
				A4_Run_P	 := FALSE;
				A_Comp		 := FALSE;
				PRO_A4_[0] := PRO_A4_[0] + 5;		 
			END_IF;
		15: // WAIT XY
			M_CHOOSE_POS_XY(DATA := 0, ID := 0, XY_CONST := TRUE);
			IF NOT A4_Run_P THEN
				A_Comp := FALSE;
				A4_Run_P := TRUE;
			END_IF		
			IF MOVP_A.Error OR MOVL_A.Error THEN
				A4_Run_L	:= FALSE;
				A4_Run_P 	:= FALSE;	 	 
			END_IF;				
			IF A_Comp AND A4_Run_P AND A_Allow_NextStep THEN
				A4_Run_L	:= FALSE;
				A4_Run_P 	:=FALSE;	
				PRO_A4_[0] := PRO_A4_[0] + 5;			 
			END_IF;
		20: // WAIT XYR
			M_CHOOSE_POS(DATA := 0, ID := 0, XYR_CONST := FALSE, Z_CONST:= TRUE);
			IF NOT A4_Run_P THEN
				A_Comp := FALSE;
				A4_Run_P := TRUE;
			END_IF		
			IF MOVP_A.Error OR MOVL_A.Error THEN
				A4_Run_L	:= FALSE;
				A4_Run_P 	:= FALSE;	 	 
			END_IF;				
			IF A_Comp AND A4_Run_P AND A_Allow_NextStep THEN
				A4_Run_L	:= FALSE;
				A4_Run_P 	:=FALSE;	
				PRO_A4_[0] := PRO_A4_[0] + 10;			 
			END_IF;
		30:
			Wait_A4_Finish := TRUE;
		
	END_CASE
ELSE
	PRO_A4_[0] := 0;
END_IF
END_ACTION

ACTION A1_Pick_T1_4:
Project_4_Delay_A1( PT := TO_TIME(GVL.Pro4_.ST_A.TDelay_pick_T1));
IF Pick_A4_T1_Run THEN
	CASE PRO_A4_[1] OF
		0: // RESET
				A4_Run_L	 := FALSE;
				A4_Run_P	 := FALSE;
				A_Comp		 := FALSE;		
				Project_4_Delay_A.IN := FALSE;	
				PRO_A4_[1] := PRO_A4_[1] + 5;
		5: // BF R PICK T1
			M_R_Mov(DATA:= 0, ID := 1, R_ := TRUE, X_ := FALSE, Y_ := FALSE, Z_ := FALSE);
			//M_CHOOSE_POS(DATA := 1, ID := 1, XYR_CONST := TRUE, Z_CONST:= FALSE); // pos 1 BF PICK 1
			IF NOT A4_Run_P THEN
				A_Comp	 := FALSE;
				A4_Run_P := TRUE;
			END_IF	
			IF MOVP_A.Error OR MOVL_A.Error THEN
				A4_Run_L	:= FALSE;
				A4_Run_P 	:= FALSE;	 
			END_IF;			
	
			IF A_Comp AND A4_Run_P AND A_Allow_NextStep THEN
				A4_Run_L	 := FALSE;
				A4_Run_P	 := FALSE;
				A_Comp		 := FALSE;
				PRO_A4_[1] := PRO_A4_[1] + 5;		 
			END_IF;			
		10: // BF Z PICK T1
			M_CHOOSE_POS(DATA := 0, ID := 1, XYR_CONST := TRUE, Z_CONST:= FALSE); // pos 1 BF PICK 1
			IF NOT A4_Run_P THEN
				A_Comp	 := FALSE;
				A4_Run_P := TRUE;
			END_IF	
			IF MOVP_A.Error OR MOVL_A.Error THEN
				A4_Run_L	:= FALSE;
				A4_Run_P 	:= FALSE;	 
			END_IF;			
	
			IF A_Comp AND A4_Run_P AND A_Allow_NextStep THEN
				A4_Run_L	 := FALSE;
				A4_Run_P	 := FALSE;
				A_Comp		 := FALSE;
				PRO_A4_[1] := PRO_A4_[1] + 10;		 
			END_IF;
	
		20: // BF XY PICK T1
			M_CHOOSE_POS(DATA := 0, ID := 1, XYR_CONST := FALSE, Z_CONST:= TRUE); // pos 1
			IF NOT A4_Run_P THEN
				A_Comp 		:= FALSE;
				A4_Run_P 	:= TRUE;
			END_IF		
			IF MOVP_A.Error OR MOVL_A.Error THEN
				A4_Run_L	:= FALSE;
				A4_Run_P    :=FALSE;	 	 
			END_IF;				
			IF A_Comp AND A4_Run_P AND A_Allow_NextStep THEN
				A4_Run_L	:= FALSE;
				A4_Run_P 	:= FALSE;	
				PRO_A4_[1] := PRO_A4_[1] + 10;		 
			END_IF;
		30: // CHECK ALLOW PICK MC1
			IF (GVL.Pro4_.Process.DATA_MC_TS = 3 OR GVL.Pro4_.Process.DATA_MC_TS = 4) AND GVL.Pro4_.Signal_In.T_Ts_Press_Up.Q THEN
			//IF TRUE THEN
				change_fac_vel_max_A := TRUE; //namnv0204
				change_fac_vel_max_A_test := TRUE;
				PRO_A4_[1] := PRO_A4_[1] + 10;	
			END_IF;	
		40: // XY PICK T1
			change_fac_vel_max_A := TRUE; //namnv0204
			M_CHOOSE_POS(DATA := 0, ID := 2, XYR_CONST := FALSE, Z_CONST:= TRUE); // pos 2
// 			IF NOT A4_Run_P THEN
			IF NOT A4_Run_P AND (GVL.Fac_Vel_Set_A = GVL.Pro4_.Auto.Fac_Vel_Max_A) THEN  //namnv0204
				A_Comp 		:= FALSE;
				A4_Run_P 	:= TRUE;
			END_IF		
			IF MOVP_A.Error OR MOVL_A.Error THEN
				A4_Run_L	:= FALSE;
				A4_Run_P    :=FALSE;	 	 
			END_IF;				
			IF A_Comp AND A4_Run_P AND A_Allow_NextStep THEN
				A4_Run_L	:= FALSE;
				A4_Run_P :=FALSE;	
				PRO_A4_[1] := PRO_A4_[1] + 10;		 
			END_IF;	
		50: // Z PICK T1
			M_CHOOSE_POS(DATA := 0, ID := 2, XYR_CONST := TRUE, Z_CONST:= FALSE); // pos 2 PICK 1
			IF (NOT GVL.Pro4_.ST_MC.Mode_Dry) THEN
				GVL.RB_A_.Tool_1 := TRUE;
			END_IF;
			IF NOT A4_Run_P THEN
				A_Comp	 := FALSE;
				A4_Run_P := TRUE;
			END_IF	
			IF MOVP_A.Error OR MOVL_A.Error THEN
				A4_Run_L	:= FALSE;
				A4_Run_P 	:= FALSE;	 
			END_IF;			
	
			IF A_Comp AND A4_Run_P AND A_Allow_NextStep THEN
				A4_Run_L	 := FALSE;
				A4_Run_P	 := FALSE;
				A_Comp		 := FALSE;
				PRO_A4_[1] := PRO_A4_[1] + 10;		 
			END_IF;
		
		60: // ON VACUUM
			IF (NOT GVL.Pro4_.ST_MC.Mode_Dry) THEN
				GVL.RB_A_.Tool_1 := TRUE;
			END_IF;
			Project_4_Delay_A1.IN := TRUE;
			IF Project_4_Delay_A1.Q AND A_Allow_NextStep AND (GVL.RB_Signal_In.SS_RBA_Tool_1.Q OR GVL.Pro4_.ST_MC.Mode_Skip_ss_T1_A) THEN
				PRO_A4_[1] := PRO_A4_[1] + 10; 	
			END_IF;
		70: // BF Z PICK T1
			Project_4_Delay_A1.IN := FALSE;
			M_CHOOSE_POS(DATA := 0, ID := 1, XYR_CONST := TRUE, Z_CONST:= FALSE); // pos 1 BF PICK 1
			IF NOT A4_Run_P THEN
				A_Comp	 := FALSE;
				A4_Run_P := TRUE;
			END_IF	
			IF MOVP_A.Error OR MOVL_A.Error THEN
				A4_Run_L	:= FALSE;
				A4_Run_P 	:= FALSE;	 
			END_IF;			
	
			IF A_Comp AND A4_Run_P AND A_Allow_NextStep THEN
				A4_Run_L	 := FALSE;
				A4_Run_P	 := FALSE;
				A_Comp		 := FALSE;
				PRO_A4_[1] := PRO_A4_[1] + 10;		 
			END_IF;
		80: // BF XY PICK T1 Namnv
// 			M_CHOOSE_POS(DATA := 1, ID := 1, XYR_CONST := FALSE, Z_CONST:= TRUE); // pos 1
			M_CHOOSE_POS(DATA := 0, ID := 1, XYR_CONST := FALSE, Z_CONST:= TRUE); // pos 1
			IF NOT A4_Run_P THEN
				A_Comp 		:= FALSE;
				A4_Run_P 	:= TRUE;
			END_IF		
			IF MOVP_A.Error OR MOVL_A.Error THEN
				A4_Run_L	:= FALSE;
				A4_Run_P    :=FALSE;	 	 
			END_IF;				
			IF A_Comp AND A4_Run_P AND A_Allow_NextStep THEN
				A4_Run_L	:= FALSE;
				A4_Run_P :=FALSE;	
				PRO_A4_[1] := PRO_A4_[1] + 10;		 
				change_fac_vel_max_A := FALSE; //namnv0204
				change_fac_vel_max_A_test := FALSE;
			END_IF
		
		90: // Done
			//  DATA_B_T1 := 3; // NG TS
			IF GVL.Pro4_.Process.DATA_MC_TS = 3 THEN
				GVL.Pro4_.Process.DATA_TOOL_A1_IN := 1;
			ELSIF GVL.Pro4_.Process.DATA_MC_TS = 4 THEN
				GVL.Pro4_.Process.DATA_TOOL_A1_IN := 3;
			END_IF;
			Project_4_Delay_A.IN := FALSE;
			Pick_A4_T1_Finish := TRUE;
			change_fac_vel_max_A := FALSE; //namnv0204
			change_fac_vel_max_A_test := FALSE;

			
			
	END_CASE
ELSE
	PRO_A4_[1] := 0;
END_IF
END_ACTION

ACTION A2_Place_T1_OK_4:
Project_4_Delay_A2(PT := TO_TIME(GVL.Pro4_.ST_A.TDelay_Place_T1)*100);
IF Place_OK_A4_T1_Run THEN
	CASE PRO_A4_[2] OF
		0: // RESET
				A4_Run_L	 := FALSE;
				A4_Run_P	 := FALSE;
				A_Comp		 := FALSE;		
				Project_4_Delay_A2.IN := FALSE;	
				PRO_A4_[2] := PRO_A4_[2] + 10;
		10: // BF Z Plcae T1  Namnv
// 			M_CHOOSE_POS(DATA := 0, ID := 4, XYR_CONST := TRUE, Z_CONST:= FALSE); // pos 3 BF Place OK 1
// 			IF NOT A4_Run_P THEN
// 				A_Comp	 := FALSE;
// 				A4_Run_P := TRUE;
// 			END_IF	
// 			IF MOVP_A.Error OR MOVL_A.Error THEN
// 				A4_Run_L	:= FALSE;
// 				A4_Run_P 	:= FALSE;	 
// 			END_IF;			
// 	
// 			IF A_Comp AND A4_Run_P AND A_Allow_NextStep THEN
// 				A4_Run_L	 := FALSE;
// 				A4_Run_P	 := FALSE;
// 				A_Comp		 := FALSE;
// 				PRO_A4_[2] := PRO_A4_[2] + 10;		 
// 			END_IF;
			
			PRO_A4_[2] := PRO_A4_[2] + 10;	
	
		20: // BF XY Place T1
			M_CHOOSE_POS(DATA := 0, ID := 4, XYR_CONST := FALSE, Z_CONST:= TRUE); // pos 3
			//IF NOT A4_Run_P THEN
			RBA_BufferMode := 5;
			IF (NOT A4_Run_P) AND (NOT A4_Run_L) THEN //namnv
				A_Comp 		:= FALSE;
				A4_Run_P 	:= TRUE;
				// namnv0304
// 				IF (GVL.Pro4_.Process.DATA_TOOL_A1_IN = 2 OR GVL.Pro4_.Process.DATA_TOOL_A1_IN = 3) AND (GVL.Pro4_.Process.DATA_TOOL_A2_OUT = 2 OR GVL.Pro4_.Process.DATA_TOOL_A2_OUT = 3) AND (Pro_A4_BF = 70) THEN
// 					A4_Run_L 	:= TRUE;
// 				ELSE
// 					A4_Run_P 	:= TRUE;
// 				END_IF
			END_IF		
			IF MOVP_A.Error OR MOVL_A.Error THEN
				A4_Run_L	:= FALSE;
				A4_Run_P    := FALSE;	 	 
			END_IF;				
			//IF A_Comp AND A4_Run_P AND A_Allow_NextStep THEN
			IF A_Comp AND (A4_Run_L OR A4_Run_P) AND A_Allow_NextStep THEN //namnv
				A4_Run_L	:= FALSE;
				A4_Run_P 	:= FALSE;	
				PRO_A4_[2] := PRO_A4_[2] + 10;		 
			END_IF;
		30: // CHECK ALLOW PICK MC2
			IF GVL.Pro4_.Process.DATA_MC_VS = 2 THEN
			//IF TRUE THEN
				PRO_A4_[2] := PRO_A4_[2] + 5;	
			END_IF;	
		35:// quay tool trước
			M_R_Mov(DATA:= 0, ID := 5, R_ := TRUE, X_ := FALSE, Y_ := FALSE, Z_ := FALSE);
			RBA_BufferMode := 5;
			IF NOT A4_Run_P THEN
				A_Comp	 := FALSE;
				A4_Run_P := TRUE;
			END_IF	
			IF MOVP_A.Error OR MOVL_A.Error THEN
				A4_Run_L	:= FALSE;
				A4_Run_P 	:= FALSE;	 
			END_IF;			
	
			IF A_Comp AND A4_Run_P AND A_Allow_NextStep THEN
				A4_Run_L	 := FALSE;
				A4_Run_P	 := FALSE;
				A_Comp		 := FALSE;
				PRO_A4_[2] := PRO_A4_[2] + 5;		 
		
			END_IF;	
		
		40: // XY Place T1
			M_CHOOSE_POS(DATA := 0, ID := 5, XYR_CONST := FALSE, Z_CONST:= TRUE); // pos 2
			RBA_BufferMode := 0;
			//IF NOT A4_Run_P THEN
			IF (NOT A4_Run_P) AND (NOT A4_Run_L) THEN //namnv
				A_Comp 		:= FALSE;
				A4_Run_P 	:= TRUE;
				// namnv
// 				IF (GVL.Pro4_.Process.DATA_TOOL_A1_IN = 2 OR GVL.Pro4_.Process.DATA_TOOL_A1_IN = 3) AND (GVL.Pro4_.Process.DATA_TOOL_A2_OUT = 2 OR GVL.Pro4_.Process.DATA_TOOL_A2_OUT = 3) AND (Pro_A4_BF = 70) THEN
// 					A4_Run_L 	:= TRUE;
// 				ELSE
// 					A4_Run_P 	:= TRUE;
// 				END_IF
			END_IF		
			IF MOVP_A.Error OR MOVL_A.Error THEN
				A4_Run_L	:= FALSE;
				A4_Run_P    := FALSE;	 	 
			END_IF;				
			//IF A_Comp AND A4_Run_P AND A_Allow_NextStep THEN
			IF A_Comp AND (A4_Run_L OR A4_Run_P) AND A_Allow_NextStep THEN //namnv
				A4_Run_L	:= FALSE;
				A4_Run_P :=FALSE;	
				PRO_A4_[2] := PRO_A4_[2] + 10;		 
			END_IF;	
		50: // Z Place T1 - Before 15mm
			M_CHOOSE_POS_Z_BF(DATA := 0, ID := 5, XYR_CONST := TRUE, Z_CONST:= FALSE); // pos 2 PICK 1
			IF NOT A4_Run_P THEN
				A_Comp	 := FALSE;
				A4_Run_P := TRUE;
			END_IF	
			IF MOVP_A.Error OR MOVL_A.Error THEN
				A4_Run_L	:= FALSE;
				A4_Run_P 	:= FALSE;	 
			END_IF;			
	
			IF A_Comp AND A4_Run_P AND A_Allow_NextStep THEN
				A4_Run_L	 := FALSE;
				A4_Run_P	 := FALSE;
				A_Comp		 := FALSE;
				PRO_A4_[2] := PRO_A4_[2] + 5;		 
			END_IF;
		55: // Z Place T1
			change_fac_vel_A := TRUE;
			M_CHOOSE_POS(DATA := 0, ID := 5, XYR_CONST := TRUE, Z_CONST:= FALSE); // pos 2 PICK 1
			IF NOT A4_Run_P AND (GVL.Fac_Vel_Set_A = GVL.Fac_Vel_Slow) THEN
				A_Comp	 := FALSE;
				A4_Run_P := TRUE;
			END_IF	
			IF MOVP_A.Error OR MOVL_A.Error THEN
				A4_Run_L	:= FALSE;
				A4_Run_P 	:= FALSE;	 
			END_IF;			
	
			IF A_Comp AND A4_Run_P AND A_Allow_NextStep THEN
				A4_Run_L	 := FALSE;
				A4_Run_P	 := FALSE;
				A_Comp		 := FALSE;
				PRO_A4_[2] := PRO_A4_[2] + 5;
				change_fac_vel_A := FALSE;		 
			END_IF;
			
		60: // ON VACUUM
			GVL.RB_A_.Tool_1 := FALSE;
			Project_4_Delay_A2.IN:= TRUE;
			IF Project_4_Delay_A2.Q AND A_Allow_NextStep  THEN
				PRO_A4_[2] := PRO_A4_[2] + 10; 	
			END_IF;
		70: // BF Z Place OK T1
			
			M_CHOOSE_POS(DATA := 0, ID := 4, XYR_CONST := TRUE, Z_CONST:= FALSE); 
			IF NOT A4_Run_P THEN
				A_Comp	 := FALSE;
				A4_Run_P := TRUE;
			END_IF	
			IF MOVP_A.Error OR MOVL_A.Error THEN
				A4_Run_L	:= FALSE;
				A4_Run_P 	:= FALSE;	 
			END_IF;			
	
			IF A_Comp AND A4_Run_P AND A_Allow_NextStep THEN
				A4_Run_L	 := FALSE;
				A4_Run_P	 := FALSE;
				A_Comp		 := FALSE;
				IF (GVL.Pro4_.Process.DATA_TOOL_A2_OUT = 2) THEN
					GVL.Pro4_.Process.DATA_TOOL_A1_IN_OLD := GVL.Pro4_.Process.DATA_TOOL_A1_IN;
					GVL.Pro4_.Process.DATA_TOOL_A1_IN := 0;
					PRO_A4_[2] := 90;
				ELSE
					PRO_A4_[2] := PRO_A4_[2] + 10;	
				END_IF
				
				 
			END_IF;
		80: // BF XY PPlace OK T1
			//M_CHOOSE_POS(DATA := 0, ID := 4, XYR_CONST := FALSE, Z_CONST:= TRUE); // pos 4
			RBA_BufferMode := 5;
			M_R_Mov(DATA:= 0, ID := 4, R_ := FALSE, X_ := TRUE, Y_ := TRUE, Z_ := FALSE);
			IF NOT A4_Run_P THEN
				A_Comp 		:= FALSE;
				A4_Run_P 	:= TRUE;
			END_IF		
			IF MOVP_A.Error OR MOVL_A.Error THEN
				A4_Run_L	:= FALSE;
				A4_Run_P    :=FALSE;	 	 
			END_IF;				
			IF A_Comp AND A4_Run_P AND A_Allow_NextStep THEN
				A4_Run_L	:= FALSE;
				A4_Run_P :=FALSE;	
				PRO_A4_[2] := PRO_A4_[2] + 5;		 
				GVL.Pro4_.Process.DATA_TOOL_A1_IN_OLD := GVL.Pro4_.Process.DATA_TOOL_A1_IN;
				GVL.Pro4_.Process.DATA_TOOL_A1_IN := 0;
			END_IF
			// namnv
			
		85:// quay tool sau
			M_R_Mov(DATA:= 0, ID := 4, R_ := TRUE, X_ := FALSE, Y_ := FALSE, Z_ := FALSE);
			IF NOT A4_Run_P THEN
				A_Comp	 := FALSE;
				A4_Run_P := TRUE;
			END_IF	
			IF MOVP_A.Error OR MOVL_A.Error THEN
				A4_Run_L	:= FALSE;
				A4_Run_P 	:= FALSE;	 
			END_IF;			
	
			IF A_Comp AND A4_Run_P AND A_Allow_NextStep THEN
				A4_Run_L	 := FALSE;
				A4_Run_P	 := FALSE;
				A_Comp		 := FALSE;
				PRO_A4_[2] := PRO_A4_[2] + 5;		 
		
			END_IF;			
		
		90: // Done
			RBA_BufferMode := 0;
			GVL.Pro4_.Process.DATA_TOOL_A1_IN := 0;
			Project_4_Delay_A2.IN := FALSE;	
			Place_OK_A4_T1_Finish := TRUE;
			
			
	END_CASE
ELSE
	PRO_A4_[2] := 0;
END_IF
END_ACTION

ACTION A3_Place_T1_NG_4:
Project_4_Delay_A(PT := TO_TIME(GVL.Pro4_.ST_A.TDelay_Place_T1)*100);
IF Place_NG_A4_T1_Run THEN
	CASE PRO_A4_[3] OF
		0: // RESET
				A4_Run_L	 := FALSE;
				A4_Run_P	 := FALSE;
				A_Comp		 := FALSE;		
				Project_4_Delay_A.IN := FALSE;	
				PRO_A4_[3] := PRO_A4_[3] + 10;
		10: // BF Z Plcae NG T1
			M_CHOOSE_POS(DATA := 0, ID := 6, XYR_CONST := TRUE, Z_CONST:= FALSE); // pos 3 BF Place OK 1
			IF NOT A4_Run_P THEN
				A_Comp	 := FALSE;
				A4_Run_P := TRUE;
			END_IF	
			IF MOVP_A.Error OR MOVL_A.Error THEN
				A4_Run_L	:= FALSE;
				A4_Run_P 	:= FALSE;	 
			END_IF;			
	
			IF A_Comp AND A4_Run_P AND A_Allow_NextStep THEN
				A4_Run_L	 := FALSE;
				A4_Run_P	 := FALSE;
				A_Comp		 := FALSE;
				PRO_A4_[3] := PRO_A4_[3] + 10;		 
			END_IF;
	
		20: // BF XY Place T1
			M_R_Mov(DATA:= 0, ID := 6, R_ := FALSE, X_ := TRUE, Y_ := TRUE, Z_ := FALSE);
			//M_CHOOSE_POS(DATA := 0, ID := 6, XYR_CONST := FALSE, Z_CONST:= TRUE); // pos 3
			IF NOT A4_Run_P THEN
				A_Comp 		:= FALSE;
				A4_Run_P 	:= TRUE;
			END_IF		
			IF MOVP_A.Error OR MOVL_A.Error THEN
				A4_Run_L	:= FALSE;
				A4_Run_P    := FALSE;	 	 
			END_IF;				
			IF A_Comp AND A4_Run_P AND A_Allow_NextStep THEN
				A4_Run_L	:= FALSE;
				A4_Run_P 	:= FALSE;	
				PRO_A4_[3] := PRO_A4_[3] + 5;		 
			END_IF;
		25: // BF XY Place T1
			M_R_Mov(DATA:= 0, ID := 6, R_ := TRUE, X_ := FALSE, Y_ := FALSE, Z_ := FALSE);
			//M_CHOOSE_POS(DATA := 0, ID := 6, XYR_CONST := FALSE, Z_CONST:= TRUE); // pos 3
			IF NOT A4_Run_P THEN
				A_Comp 		:= FALSE;
				A4_Run_P 	:= TRUE;
			END_IF		
			IF MOVP_A.Error OR MOVL_A.Error THEN
				A4_Run_L	:= FALSE;
				A4_Run_P    := FALSE;	 	 
			END_IF;				
			IF A_Comp AND A4_Run_P AND A_Allow_NextStep THEN
				A4_Run_L	:= FALSE;
				A4_Run_P 	:= FALSE;	
				PRO_A4_[3] := PRO_A4_[3] + 5;		 
			END_IF;			
	
		30: // CHECK ALLOW PLACE CNV NG TS
			IF ALLOW_PLACE_CNV_NG_TS THEN
				PRO_A4_[3] := PRO_A4_[3] + 10;	
			END_IF;	
		40: // XY Place NG T1
			M_CHOOSE_POS(DATA := 0, ID := 7, XYR_CONST := FALSE, Z_CONST:= TRUE); // pos 2
			IF NOT A4_Run_P THEN
				A_Comp 		:= FALSE;
				A4_Run_P 	:= TRUE;
			END_IF		
			IF MOVP_A.Error OR MOVL_A.Error THEN
				A4_Run_L	:= FALSE;
				A4_Run_P    := FALSE;	 	 
			END_IF;				
			IF A_Comp AND A4_Run_P AND A_Allow_NextStep THEN
				A4_Run_L	:= FALSE;
				A4_Run_P :=FALSE;	
				PRO_A4_[3] := PRO_A4_[3] + 10;		 
			END_IF;	
		50: // Z Place T1
			M_CHOOSE_POS(DATA := 0, ID := 7, XYR_CONST := TRUE, Z_CONST:= FALSE); // pos 2 PICK 1
			IF NOT A4_Run_P THEN
				A_Comp	 := FALSE;
				A4_Run_P := TRUE;
			END_IF	
			IF MOVP_A.Error OR MOVL_A.Error THEN
				A4_Run_L	:= FALSE;
				A4_Run_P 	:= FALSE;	 
			END_IF;			
	
			IF A_Comp AND A4_Run_P AND A_Allow_NextStep THEN
				A4_Run_L	 := FALSE;
				A4_Run_P	 := FALSE;
				A_Comp		 := FALSE;
				PRO_A4_[3] := PRO_A4_[3] + 10;		 
			END_IF;
		
		60: // OFF VACUUM
			GVL.RB_A_.Tool_1 := FALSE;
			Project_4_Delay_A.IN:= TRUE;
			IF Project_4_Delay_A.Q AND A_Allow_NextStep  THEN
				PRO_A4_[3] := PRO_A4_[3] + 10; 	
			END_IF;
		70: // BF Z Place NG T1
			M_CHOOSE_POS(DATA := 0, ID := 6, XYR_CONST := TRUE, Z_CONST:= FALSE); 
			IF NOT A4_Run_P THEN
				A_Comp	 := FALSE;
				A4_Run_P := TRUE;
			END_IF	
			IF MOVP_A.Error OR MOVL_A.Error THEN
				A4_Run_L	:= FALSE;
				A4_Run_P 	:= FALSE;	 
			END_IF;			
	
			IF A_Comp AND A4_Run_P AND A_Allow_NextStep THEN
				A4_Run_L	 := FALSE;
				A4_Run_P	 := FALSE;
				A_Comp		 := FALSE;
				PRO_A4_[3] := PRO_A4_[3] + 10;		 
			END_IF;
		80: // BF XY PPlace NG T1
			M_CHOOSE_POS(DATA := 0, ID := 6, XYR_CONST := FALSE, Z_CONST:= TRUE); // pos 4
			IF NOT A4_Run_P THEN
				A_Comp 		:= FALSE;
				A4_Run_P 	:= TRUE;
			END_IF		
			IF MOVP_A.Error OR MOVL_A.Error THEN
				A4_Run_L	:= FALSE;
				A4_Run_P    := FALSE;	 	 
			END_IF;				
			IF A_Comp AND A4_Run_P AND A_Allow_NextStep THEN
				A4_Run_L	:= FALSE;
				A4_Run_P    := FALSE;	
				PRO_A4_[3] := PRO_A4_[3] + 10;		 
			END_IF
		
		90: // Done
			GVL.Pro4_.Process.DATA_TOOL_A1_IN := 0;
			Project_4_Delay_A.IN := FALSE;	
			Place_NG_A4_T1_Finish    := TRUE;
			
			
	END_CASE
ELSE
	PRO_A4_[3] := 0;
END_IF
END_ACTION

ACTION A4_Pick_T2_4:
Project_4_Delay_A4(PT := TO_TIME(GVL.Pro4_.ST_A.TDelay_pick_T2)*100);
Ton_tacktime(PT := T#1000000MS);
IF Pick_A4_T2_Run THEN
	CASE PRO_A4_[4] OF
		0: // RESET
				A4_Run_L	 := FALSE;
				A4_Run_P	 := FALSE;
				A_Comp		 := FALSE;		
				Project_4_Delay_A4.IN := FALSE;	
				PRO_A4_[4] := PRO_A4_[4] + 5;
		5: // BF R PICK T1
			M_R_Mov(DATA:= 0, ID := 8, R_ := TRUE, X_ := FALSE, Y_ := FALSE, Z_ := FALSE);
			//M_CHOOSE_POS(DATA := 1, ID := 1, XYR_CONST := TRUE, Z_CONST:= FALSE); // pos 1 BF PICK 1
// 			IF NOT A4_Run_P THEN
// 				A_Comp	 := FALSE;
// 				A4_Run_P := TRUE;
// 			END_IF	
// 			IF MOVP_A.Error OR MOVL_A.Error THEN
// 				A4_Run_L	:= FALSE;
// 				A4_Run_P 	:= FALSE;	 
// 			END_IF;			
// 	
// 			IF A_Comp AND A4_Run_P AND A_Allow_NextStep THEN
// 				A4_Run_L	 := FALSE;
// 				A4_Run_P	 := FALSE;
// 				A_Comp		 := FALSE;
// 				PRO_A4_[4] := PRO_A4_[4] + 5;		 
// 				
// 				IF GVL.Pro4_.Process.DATA_TOOL_A1_IN = 2 OR GVL.Pro4_.Process.DATA_TOOL_A1_IN = 3 THEN  // namnv
// 					PRO_A4_[4] := 30;
// 				END_IF
// 			END_IF;			
			PRO_A4_[4] := PRO_A4_[4] + 5;		 
				
		10: // BF Z PICK T2
// 			M_CHOOSE_POS(DATA := 0, ID := 8, XYR_CONST := TRUE, Z_CONST:= FALSE); // pos 1 BF PICK 1
// 			IF NOT A4_Run_P THEN
// 				A_Comp	 := FALSE;
// 				A4_Run_P := TRUE;
// 			END_IF	
// 			IF MOVP_A.Error OR MOVL_A.Error THEN
// 				A4_Run_L	:= FALSE;
// 				A4_Run_P 	:= FALSE;	 
// 			END_IF;			
// 	
// 			IF A_Comp AND A4_Run_P AND A_Allow_NextStep THEN
// 				A4_Run_L	 := FALSE;
// 				A4_Run_P	 := FALSE;
// 				A_Comp		 := FALSE;
// 				PRO_A4_[4] := PRO_A4_[4] + 10;		 
// 			END_IF;
			PRO_A4_[4] := PRO_A4_[4] + 10;	//Namnv
		20: // BF XY PICK T2
			M_CHOOSE_POS(DATA := 0, ID := 8, XYR_CONST := FALSE, Z_CONST:= TRUE); // pos 1
			IF NOT A4_Run_P THEN
				A_Comp 		:= FALSE;
				A4_Run_P 	:= TRUE;
			END_IF		
			IF MOVP_A.Error OR MOVL_A.Error THEN
				A4_Run_L	:= FALSE;
				A4_Run_P    :=FALSE;	 	 
			END_IF;				
			IF A_Comp AND A4_Run_P AND A_Allow_NextStep THEN
				A4_Run_L	:= FALSE;
				A4_Run_P :=FALSE;	
				PRO_A4_[4] := PRO_A4_[4] + 10;		 
			END_IF;
		30: // CHECK ALLOW PICK MC2
			//IF GVL.Pro4_.Process.DATA_MC_VS = 3 OR GVL.Pro4_.Process.DATA_MC_VS = 4 THEN
			//namnv
			IF GVL.Pro4_.Process.DATA_MC_VS = 3 OR GVL.Pro4_.Process.DATA_MC_VS = 4 OR GVL.Pro4_.Process.DATA_MC_VS = 5 THEN	
			//IF TRUE THEN
				PRO_A4_[4] := PRO_A4_[4] + 10;	
			END_IF;	
		40: // XY PICK T2
			M_CHOOSE_POS(DATA := 0, ID := 9, XYR_CONST := FALSE, Z_CONST:= TRUE); // pos 2
			IF NOT A4_Run_P THEN
				A_Comp 		:= FALSE;
				A4_Run_P 	:= TRUE;
			END_IF		
			IF MOVP_A.Error OR MOVL_A.Error THEN
				A4_Run_L	:= FALSE;
				A4_Run_P    :=FALSE;	 	 
			END_IF;				
			IF A_Comp AND A4_Run_P AND A_Allow_NextStep THEN
				A4_Run_L	:= FALSE;
				A4_Run_P :=FALSE;	
				PRO_A4_[4] := PRO_A4_[4] + 10;		 
			END_IF;	
		50: // Z PICK T2
			M_CHOOSE_POS(DATA := 0, ID := 9, XYR_CONST := TRUE, Z_CONST:= FALSE); // pos 2 PICK 1
			IF (NOT GVL.Pro4_.ST_MC.Mode_Dry) THEN
				GVL.RB_A_.Tool_2 := TRUE;
			END_IF;
			IF NOT A4_Run_P THEN
				A_Comp	 := FALSE;
				A4_Run_P := TRUE;
			END_IF	
			IF MOVP_A.Error OR MOVL_A.Error THEN
				A4_Run_L	:= FALSE;
				A4_Run_P 	:= FALSE;	 
			END_IF;			
	
			IF A_Comp AND A4_Run_P AND A_Allow_NextStep THEN
				A4_Run_L	 := FALSE;
				A4_Run_P	 := FALSE;
				A_Comp		 := FALSE;
				PRO_A4_[4] := PRO_A4_[4] + 10;
				GVL.Pro4_.Auto.T_tacktime_pre := GVL.Pro4_.Auto.T_tacktime_cr;
				GVL.Pro4_.Auto.T_tacktime_cr := TO_INT(Ton_tacktime.ET)/10;
				Ton_tacktime.IN := FALSE; 
				//namnv1104
				Monitor_Production.Pulse_In_ := FALSE;
				Monitor_Production.Pulse_Out_ := TRUE;
			END_IF;
		
		60: // ON VACUUM
			IF (NOT GVL.Pro4_.ST_MC.Mode_Dry) THEN
				GVL.RB_A_.Tool_2 := TRUE;
			END_IF;
			Project_4_Delay_A4.IN:= TRUE;
			IF Project_4_Delay_A4.Q AND A_Allow_NextStep AND (GVL.RB_Signal_In.SS_RBA_Tool_2.Q OR GVL.Pro4_.ST_MC.Mode_Skip_ss_T2_A) THEN
				PRO_A4_[4] := PRO_A4_[4] + 10; 	
				Ton_tacktime.IN := TRUE;
				//namnv1104
				Monitor_Production.Pulse_In_ := TRUE;
				Monitor_Production.Pulse_Out_ := FALSE;
			END_IF;
		70: // BF Z PICK T2
			Project_4_Delay_A4.IN:= FALSE;
			M_CHOOSE_POS(DATA := 0, ID := 8, XYR_CONST := TRUE, Z_CONST:= FALSE); // pos 1 BF PICK 1
			IF NOT A4_Run_P THEN
				A_Comp	 := FALSE;
				A4_Run_P := TRUE;
			END_IF	
			IF MOVP_A.Error OR MOVL_A.Error THEN
				A4_Run_L	:= FALSE;
				A4_Run_P 	:= FALSE;	 
			END_IF;			
	
			IF A_Comp AND A4_Run_P AND A_Allow_NextStep THEN
				A4_Run_L	 := FALSE;
				A4_Run_P	 := FALSE;
				A_Comp		 := FALSE;
				PRO_A4_[4] := PRO_A4_[4] + 10;		 
				
				// namnv
				IF (GVL.Pro4_.Process.DATA_TOOL_A1_IN = 2 OR GVL.Pro4_.Process.DATA_TOOL_A1_IN = 3) AND (GVL.Pro4_.Process.DATA_MC_VS = 3 OR GVL.Pro4_.Process.DATA_MC_VS = 4) THEN
					PRO_A4_[4] := 90;
				END_IF
			END_IF;
		80: // BF XY PICK T2
			M_CHOOSE_POS(DATA := 0, ID := 8, XYR_CONST := FALSE, Z_CONST:= TRUE); // pos 1
			IF NOT A4_Run_P THEN
				A_Comp 		:= FALSE;
				A4_Run_P 	:= TRUE;
			END_IF		
			IF MOVP_A.Error OR MOVL_A.Error THEN
				A4_Run_L	:= FALSE;
				A4_Run_P    :=FALSE;	 	 
			END_IF;				
			IF A_Comp AND A4_Run_P AND A_Allow_NextStep THEN
				A4_Run_L	:= FALSE;
				A4_Run_P :=FALSE;	
				PRO_A4_[4] := PRO_A4_[4] + 10;		 
			END_IF
		
		90: // Done
			//GVL.Pro4_.Process.DATA_TOOL_A2_OUT := 2;
			IF GVL.Pro4_.Process.DATA_MC_VS = 3 THEN
				GVL.Pro4_.Process.DATA_TOOL_A2_OUT := 2;
			ELSIF GVL.Pro4_.Process.DATA_MC_VS = 4 THEN
				GVL.Pro4_.Process.DATA_TOOL_A2_OUT := 3;
			END_IF;			
			//namnv - Tool2 gap hang NG test song
			IF GVL.Pro4_.Process.DATA_MC_VS = 5 THEN
				GVL.Pro4_.Process.DATA_TOOL_A2_OUT := 4;
			END_IF
			Project_4_Delay_A4.IN := FALSE;
			Pick_A4_T2_Finish := TRUE;

			
			
	END_CASE
ELSE
	PRO_A4_[4] := 0;
END_IF
END_ACTION

ACTION A5_Place_T2_OK_4:
Project_4_Delay_A5(PT := TO_TIME(GVL.Pro4_.ST_A.Tdelay_Place_T2)*100);
IF Place_OK_A4_T2_Run THEN
	CASE PRO_A4_[5] OF
		0: // RESET
				A4_Run_L	 := FALSE;
				A4_Run_P	 := FALSE;
				A_Comp		 := FALSE;		
				Project_4_Delay_A5.IN := FALSE;	
				PRO_A4_[5] := PRO_A4_[5] + 10;
		10: // BF Z Plcae T2
			M_CHOOSE_POS(DATA := 0, ID := 10, XYR_CONST := TRUE, Z_CONST:= FALSE); // pos 3 BF Place OK 1
			IF NOT A4_Run_P THEN
				A_Comp	 := FALSE;
				A4_Run_P := TRUE;
			END_IF	
			IF MOVP_A.Error OR MOVL_A.Error THEN
				A4_Run_L	:= FALSE;
				A4_Run_P 	:= FALSE;	 
			END_IF;			
	
			IF A_Comp AND A4_Run_P AND A_Allow_NextStep THEN
				A4_Run_L	 := FALSE;
				A4_Run_P	 := FALSE;
				A_Comp		 := FALSE;
				PRO_A4_[5] := PRO_A4_[5] + 5;		 
			END_IF;
		15:// XY PLACE OK T2
			M_R_Mov(DATA:= 0, ID := 10, R_ := FALSE, X_ := TRUE, Y_ := TRUE, Z_ := FALSE);
			IF NOT A4_Run_P THEN
				A_Comp 		:= FALSE;
				A4_Run_P 	:= TRUE;
			END_IF		
			IF MOVP_A.Error OR MOVL_A.Error THEN
				A4_Run_L	:= FALSE;
				A4_Run_P    :=FALSE;	 	 
			END_IF;				
			IF A_Comp AND A4_Run_P AND A_Allow_NextStep THEN
				A4_Run_L	:= FALSE;
				A4_Run_P :=FALSE;	
				PRO_A4_[5] := PRO_A4_[5] + 5;		 
			END_IF
		
		20: // BF XY Place T2
			M_CHOOSE_POS(DATA := 0, ID := 10, XYR_CONST := FALSE, Z_CONST:= TRUE); // pos 3
			IF NOT A4_Run_P THEN
				A_Comp 		:= FALSE;
				A4_Run_P 	:= TRUE;
			END_IF		
			IF MOVP_A.Error OR MOVL_A.Error THEN
				A4_Run_L	:= FALSE;
				A4_Run_P    := FALSE;	 	 
			END_IF;				
			IF A_Comp AND A4_Run_P AND A_Allow_NextStep THEN
				A4_Run_L	:= FALSE;
				A4_Run_P 	:= FALSE;	
				PRO_A4_[5] := PRO_A4_[5] + 10;		 
			END_IF;
		30: // CHECK ALLOW place OK 2 
			IF ALLOW_PLACE_CNV_OK THEN
				PRO_A4_[5] := PRO_A4_[5] + 10;	
			END_IF;	
		40: // XY Place T2
			M_CHOOSE_POS(DATA := 0, ID := 11, XYR_CONST := FALSE, Z_CONST:= TRUE); // pos 2
			IF NOT A4_Run_P THEN
				A_Comp 		:= FALSE;
				A4_Run_P 	:= TRUE;
			END_IF		
			IF MOVP_A.Error OR MOVL_A.Error THEN
				A4_Run_L	:= FALSE;
				A4_Run_P    := FALSE;	 	 
			END_IF;				
			IF A_Comp AND A4_Run_P AND A_Allow_NextStep THEN
				A4_Run_L	:= FALSE;
				A4_Run_P :=FALSE;	
				PRO_A4_[5] := PRO_A4_[5] + 10;		 
			END_IF;	
		50: // Z Place T2
			M_CHOOSE_POS(DATA := 0, ID := 11, XYR_CONST := TRUE, Z_CONST:= FALSE); // pos 2 PICK 1
			IF NOT A4_Run_P THEN
// 				A_Comp	 := FALSE;
// 				A4_Run_P := TRUE;
				IF GVL.Pro4_.Signal_In.T_Cv_OK_out.Q THEN
					A_Comp	 := FALSE;
					A4_Run_P := TRUE;
				END_IF;
			END_IF	
			IF MOVP_A.Error OR MOVL_A.Error THEN
				A4_Run_L	:= FALSE;
				A4_Run_P 	:= FALSE;	 
			END_IF;			
	
			IF A_Comp AND A4_Run_P AND A_Allow_NextStep THEN
				A4_Run_L	 := FALSE;
				A4_Run_P	 := FALSE;
				A_Comp		 := FALSE;
				PRO_A4_[5] := PRO_A4_[5] + 10;		 
			END_IF;
		
		60: // OFF VACUUM
			GVL.RB_A_.Tool_2 := FALSE;
			Project_4_Delay_A5.IN:= TRUE;
			IF Project_4_Delay_A5.Q AND A_Allow_NextStep  THEN
				PRO_A4_[5] := PRO_A4_[5] + 10; 	
			END_IF;
		70: // BF Z Place OK T2
			Project_4_Delay_A5.IN:= FALSE;
			M_CHOOSE_POS(DATA := 0, ID := 10, XYR_CONST := TRUE, Z_CONST:= FALSE); 
			IF NOT A4_Run_P THEN
				A_Comp	 := FALSE;
				A4_Run_P := TRUE;
			END_IF	
			IF MOVP_A.Error OR MOVL_A.Error THEN
				A4_Run_L	:= FALSE;
				A4_Run_P 	:= FALSE;	 
			END_IF;			
	
			IF A_Comp AND A4_Run_P AND A_Allow_NextStep THEN
				A4_Run_L	 := FALSE;
				A4_Run_P	 := FALSE;
				A_Comp		 := FALSE;
				PRO_A4_[5] := PRO_A4_[5] + 10;		 
			END_IF;
		80: // BF XY PPlace OK T2
// 			M_CHOOSE_POS(DATA := 0, ID := 10, XYR_CONST := FALSE, Z_CONST:= TRUE); // 
// 			IF NOT A4_Run_P THEN
// 				A_Comp 		:= FALSE;
// 				A4_Run_P 	:= TRUE;
// 			END_IF		
// 			IF MOVP_A.Error OR MOVL_A.Error THEN
// 				A4_Run_L	:= FALSE;
// 				A4_Run_P    :=FALSE;	 	 
// 			END_IF;				
// 			IF A_Comp AND A4_Run_P AND A_Allow_NextStep THEN
// 				A4_Run_L	:= FALSE;
// 				A4_Run_P 	:= FALSE;	
// 				PRO_A4_[5] := PRO_A4_[5] + 10;		 
// 			END_IF
			PRO_A4_[5] := PRO_A4_[5] + 10;
		90: // Done
			GVL.Pro4_.Process.DATA_TOOL_A2_OUT := 0;
			Project_4_Delay_A5.IN := FALSE;	
			Place_OK_A4_T2_Finish := TRUE;
			
			
	END_CASE
ELSE
	PRO_A4_[5] := 0;
END_IF
END_ACTION

ACTION A6_Place_T2_NG_4:
Project_4_Delay_A6(PT := TO_TIME(GVL.Pro4_.ST_A.Tdelay_Place_T2)*100);
IF Place_NG_A4_T2_Run THEN
	CASE PRO_A4_[6] OF
		0: // RESET
				A4_Run_L	 := FALSE;
				A4_Run_P	 := FALSE;
				A_Comp		 := FALSE;		
				Project_4_Delay_A6.IN := FALSE;	
				PRO_A4_[6] := PRO_A4_[6] + 10;
		10: // BF Z Plcae NG T2
			M_CHOOSE_POS(DATA := 0, ID := 12, XYR_CONST := TRUE, Z_CONST:= FALSE); // pos 3 BF Place OK 1
			IF NOT A4_Run_P THEN
				A_Comp	 := FALSE;
				A4_Run_P := TRUE;
			END_IF	
			IF MOVP_A.Error OR MOVL_A.Error THEN
				A4_Run_L	:= FALSE;
				A4_Run_P 	:= FALSE;	 
			END_IF;			
	
			IF A_Comp AND A4_Run_P AND A_Allow_NextStep THEN
				A4_Run_L	 := FALSE;
				A4_Run_P	 := FALSE;
				A_Comp		 := FALSE;
				PRO_A4_[6] := PRO_A4_[6] + 10;		 
			END_IF;
	
		20: // BF XY Place T2
			M_CHOOSE_POS(DATA := 0, ID := 12, XYR_CONST := FALSE, Z_CONST:= TRUE); // pos 3
			IF NOT A4_Run_P THEN
				A_Comp 		:= FALSE;
				A4_Run_P 	:= TRUE;
			END_IF		
			IF MOVP_A.Error OR MOVL_A.Error THEN
				A4_Run_L	:= FALSE;
				A4_Run_P    := FALSE;	 	 
			END_IF;				
			IF A_Comp AND A4_Run_P AND A_Allow_NextStep THEN
				A4_Run_L	:= FALSE;
				A4_Run_P 	:= FALSE;	
				PRO_A4_[6] := PRO_A4_[6] + 10;		 
			END_IF;
		30: // CHECK ALLOW PLACE CNV NG VS
			IF ALLOW_PLACE_CNV_NG_VS THEN
				PRO_A4_[6] := PRO_A4_[6] + 10;	
			END_IF;	
		40: // XY Place NG T2
			M_CHOOSE_POS(DATA := 0, ID := 13, XYR_CONST := FALSE, Z_CONST:= TRUE); // pos 2
			IF NOT A4_Run_P THEN
				A_Comp 		:= FALSE;
				A4_Run_P 	:= TRUE;
			END_IF		
			IF MOVP_A.Error OR MOVL_A.Error THEN
				A4_Run_L	:= FALSE;
				A4_Run_P    := FALSE;	 	 
			END_IF;				
			IF A_Comp AND A4_Run_P AND A_Allow_NextStep THEN
				A4_Run_L	:= FALSE;
				A4_Run_P :=FALSE;	
				PRO_A4_[6] := PRO_A4_[6] + 10;		 
			END_IF;	
		50: // Z Place T2
			M_CHOOSE_POS(DATA := 0, ID := 13, XYR_CONST := TRUE, Z_CONST:= FALSE); // pos 2 PICK 1
			IF NOT A4_Run_P THEN
				IF NOT GVL.Pro4_.Signal_In.T_Cv_NG_out_1.Q AND NOT GVL.Pro4_.Signal_In.T_Cv_NG_out_2.Q AND NOT GVL.Pro4_.Signal_In.T_Cv_NG_out_full.Q THEN
					A_Comp	 := FALSE;
					A4_Run_P := TRUE;
				END_IF;
			END_IF	
			IF MOVP_A.Error OR MOVL_A.Error THEN
				A4_Run_L	:= FALSE;
				A4_Run_P 	:= FALSE;	 
			END_IF;			
	
			IF A_Comp AND A4_Run_P AND A_Allow_NextStep THEN
				A4_Run_L	 := FALSE;
				A4_Run_P	 := FALSE;
				A_Comp		 := FALSE;
				PRO_A4_[6] := PRO_A4_[6] + 10;		 
			END_IF;
		
		60: // OFF VACUUM
			// namnv0104
			IF NOT GVL.Pro4_.Signal_In.T_Cv_NG_out_1.Q THEN
				GVL.RB_A_.Tool_2 := FALSE;
				Project_4_Delay_A6.IN:= TRUE;
			END_IF;
			IF Project_4_Delay_A6.Q AND A_Allow_NextStep  THEN
				PRO_A4_[6] := PRO_A4_[6] + 10; 	
			END_IF;
			
		70: // BF Z Place NG T1
			M_CHOOSE_POS(DATA := 0, ID := 12, XYR_CONST := TRUE, Z_CONST:= FALSE); 
			IF NOT A4_Run_P THEN
				A_Comp	 := FALSE;
				A4_Run_P := TRUE;
			END_IF	
			IF MOVP_A.Error OR MOVL_A.Error THEN
				A4_Run_L	:= FALSE;
				A4_Run_P 	:= FALSE;	 
			END_IF;			
	
			IF A_Comp AND A4_Run_P AND A_Allow_NextStep THEN
				A4_Run_L	 := FALSE;
				A4_Run_P	 := FALSE;
				A_Comp		 := FALSE;
				PRO_A4_[6] := PRO_A4_[6] + 10;		 
			END_IF;
		80: // BF XY PPlace NG T2
			M_CHOOSE_POS(DATA := 0, ID := 12, XYR_CONST := FALSE, Z_CONST:= TRUE); // 
			IF NOT A4_Run_P THEN
				A_Comp 		:= FALSE;
				A4_Run_P 	:= TRUE;
			END_IF		
			IF MOVP_A.Error OR MOVL_A.Error THEN
				A4_Run_L	:= FALSE;
				A4_Run_P    := FALSE;	 	 
			END_IF;				
			IF A_Comp AND A4_Run_P AND A_Allow_NextStep THEN
				A4_Run_L	:= FALSE;
				A4_Run_P    := FALSE;	
				PRO_A4_[6] := PRO_A4_[6] + 10;		 
			END_IF
		
		90: // Done
			GVL.Pro4_.Process.DATA_TOOL_A2_OUT := 0;
			Project_4_Delay_A6.IN := FALSE;	
			Place_NG_A4_T2_Finish    := TRUE;
			
			
	END_CASE
ELSE
	PRO_A4_[6] := 0;
END_IF
END_ACTION

ACTION A7_Barcode_T1_4:
//Project_4_Delay_A7(PT := TO_TIME(GVL.Pro4_.ST_MC.Delay_Trigger_Barcode_Vs)*100);
T_Wait_Trigger_Bar_VS( PT := TO_TIME(GVL.Pro4_.ST_MC.Delay_Trigger_Barcode_Vs)*100);
IF Barcode_A4_Run THEN
	CASE PRO_A4_[7] OF
		0: // RESET
				A4_Run_L	 := FALSE;
				A4_Run_P	 := FALSE;
				A_Comp		 := FALSE;			
				count_Vs := 0; // namnv
				PRO_A4_[7] := PRO_A4_[7] + 10;
		10: // XY barcode
			M_CHOOSE_POS(DATA := 0, ID := 3, XYR_CONST := FALSE, Z_CONST:= TRUE); // pos 4 barcode
			IF NOT A4_Run_P THEN
				A_Comp := FALSE;
				A4_Run_P := TRUE;
			END_IF		
			IF MOVP_A.Error OR MOVL_A.Error THEN
				A4_Run_L	:= FALSE;
				A4_Run_P 	:= FALSE;	 
			END_IF;				
			IF A_Comp AND A4_Run_P AND A_Allow_NextStep THEN
				A4_Run_L	 := FALSE;
				A4_Run_P	 := FALSE;
				A_Comp		 := FALSE;
				PRO_A4_[7] := PRO_A4_[7] + 10;		 
			END_IF;
	
		20: // Barcode Z
			M_CHOOSE_POS(DATA := 0, ID := 3, XYR_CONST := TRUE, Z_CONST:= FALSE); // pos 4 barcode
			IF NOT A4_Run_P THEN
				A_Comp := FALSE;
				A4_Run_P := TRUE;
			END_IF		
			IF MOVP_A.Error OR MOVL_A.Error THEN
				A3_Run_L	:= FALSE;
				A3_Run_P :=FALSE;	 	 
			END_IF;				
			IF A_Comp AND A4_Run_P AND A_Allow_NextStep THEN
				A4_Run_L	:= FALSE;
				A4_Run_P :=FALSE;	
				PRO_A4_[7] := PRO_A4_[7] + 10;		 
			END_IF;
	
		30: // Trigger Barcode
			// Ontrigger
			CASE D_Barcode_Vs OF
				0:
					IF GVL.Pro4_.ST_MC.Mode_Skip_Barcode_vs THEN
						D_Barcode_Vs:= 30;
					ELSE
							//GVL.Pro4_.Auto.Trigger_Barcode_Vs_On_Off := 1;
						// namnv
						GVL.Pro4_.Auto.Trigger_Barcode_Vs_On_Off := TRUE;
						//Project_4_Delay_A7.IN := TRUE;
						//IF GVL.Pro4_.Auto.Trigger_Barcode_Vs_On_Off = 1 AND Project_4_Delay_A7.q THEN
						// namnv
						//IF GVL.Pro4_.Auto.Trigger_Barcode_Vs_On_Off AND Project_4_Delay_A7.q THEN
						IF GVL.Pro4_.Auto.Trigger_Barcode_Vs_On_Off AND GVL.Pro4_.Signal_In.T_Vs_detect.Q THEN
							D_Barcode_Vs := D_Barcode_Vs +10;
						END_IF	
					END_IF	
				10:
					//Project_4_Delay_A7.IN := FALSE;
					//GVL.Pro4_.Auto.Trigger_Barcode_Vs_On_Off := 0;
					// namnv
					GVL.Pro4_.Auto.Trigger_Barcode_Vs_On_Off := FALSE;
					//IF GVL.Pro4_.Auto.Trigger_Barcode_Vs_On_Off = 0 THEN
					IF NOT GVL.Pro4_.Auto.Trigger_Barcode_Vs_On_Off THEN
						count_Vs := count_Vs +1;
						D_Barcode_Vs := D_Barcode_Vs +10;
						T_Wait_Trigger_Bar_VS.IN := TRUE;
					END_IF
				20:
					IF GVL.Pro4_.Signal_In.T_Vs_Result_Scanner.Q OR  GVL.X[30] THEN
						D_Barcode_Vs := D_Barcode_Vs +10;
						T_Wait_Trigger_Bar_VS.IN := FALSE;
					ELSIF NOT GVL.Pro4_.Signal_In.T_Ts_Result_Scanner.Q AND NOT GVL.X[30]  AND count_Vs <= 5 AND T_Wait_Trigger_Bar_VS.Q THEN
						D_Barcode_Vs := 0;
						T_Wait_Trigger_Bar_VS.IN := FALSE;
					END_IF
				30:
					GVL.Pro4_.Auto.Alarm_Not_barcode_VS := FALSE;
					// ok barcode vs
			END_CASE;
			IF count_Vs > 5 AND (GVL.X[8] OR gvl.Pro4_.Process.Re_Trigger_Barcode_Vs) THEN
				count_Vs := 0;
				GVL.Pro4_.Auto.Alarm_Not_barcode_VS := FALSE;
			END_IF
			
			IF count_Vs > 5 AND D_Barcode_Vs = 20 AND NOT GVL.Pro4_.Auto.Alarm_Not_barcode_VS  THEN
				GVL.Pro4_.Auto.Alarm_Not_barcode_VS := TRUE;
				PRO_A4_[7] := PRO_A4_[7] + 10; 	
			END_IF
			
			IF D_Barcode_Vs = 30 AND A_Allow_NextStep  THEN
				GVL.Pro4_.Auto.Alarm_Not_barcode_VS := FALSE;
				count_Vs := 0;
				PRO_A4_[7] := PRO_A4_[7] + 10; 	
			END_IF;
			
		40: // Z WAIT
			D_Barcode_vs := 0;
			
			M_CHOOSE_POS(DATA := 0, ID := 0, XYR_CONST := TRUE, Z_CONST:= FALSE); // pos wait
			IF NOT A4_Run_P THEN
				A_Comp := FALSE;
				A4_Run_P := TRUE;
			END_IF		
			IF MOVP_A.Error OR MOVL_A.Error THEN
				A4_Run_L	:= FALSE;
				A4_Run_P 	:= FALSE;	 
			END_IF;				
			IF A_Comp AND A4_Run_P AND A_Allow_NextStep THEN
				A4_Run_L	 := FALSE;
				A4_Run_P	 := FALSE;
				A_Comp		 := FALSE;
				PRO_A4_[7] := PRO_A4_[7] + 10;		 
			END_IF;		
		50:
			// GVL.Pro4_.Process.DATA_TOOL_A1_IN := 3;
			// namnv - Doc barcode xong cho du lieu A_T1 = 2 (OK)
			IF (GVL.Pro4_.Auto.Alarm_Not_barcode_VS) THEN
				GVL.Pro4_.Process.DATA_TOOL_A1_IN := 2;
			ELSE
				GVL.Pro4_.Process.DATA_TOOL_A1_IN := 2;
			END_IF
			GVL.Pro4_.Auto.Alarm_Not_barcode_VS := FALSE;
			//GVL.Pro4_.Process.DATA_TOOL_A1_IN := 2;
			Barcode_A4_Finish := TRUE;
			
			
	END_CASE
ELSE
	PRO_A4_[7] := 0;
END_IF
END_ACTION

ACTION A8_Place_T2_NG_TS_4:
Project_4_Delay_A8(PT := TO_TIME(GVL.Pro4_.ST_A.Tdelay_Place_T2)*100);
IF Place_NG_TS_A4_T2_Run THEN
	CASE PRO_A4_[8] OF
		0: // RESET
				A4_Run_L	 := FALSE;
				A4_Run_P	 := FALSE;
				A_Comp		 := FALSE;		
				Project_4_Delay_A8.IN := FALSE;	
				PRO_A4_[8] := PRO_A4_[8] + 10;
		10: // BF Z Plcae NG T2
			M_CHOOSE_POS(DATA := 0, ID := 6, XYR_CONST := TRUE, Z_CONST:= FALSE); // pos 3 BF Place OK 1
			IF NOT A4_Run_P THEN
				A_Comp	 := FALSE;
				A4_Run_P := TRUE;
			END_IF	
			IF MOVP_A.Error OR MOVL_A.Error THEN
				A4_Run_L	:= FALSE;
				A4_Run_P 	:= FALSE;	 
			END_IF;			
	
			IF A_Comp AND A4_Run_P AND A_Allow_NextStep THEN
				A4_Run_L	 := FALSE;
				A4_Run_P	 := FALSE;
				A_Comp		 := FALSE;
				PRO_A4_[8] := PRO_A4_[8] + 10;		 
			END_IF;
	
		20: // BF XY Place T2
			M_CHOOSE_POS(DATA := 0, ID := 6, XYR_CONST := FALSE, Z_CONST:= TRUE); // pos 3
			IF NOT A4_Run_P THEN
				A_Comp 		:= FALSE;
				A4_Run_P 	:= TRUE;
			END_IF		
			IF MOVP_A.Error OR MOVL_A.Error THEN
				A4_Run_L	:= FALSE;
				A4_Run_P    := FALSE;	 	 
			END_IF;				
			IF A_Comp AND A4_Run_P AND A_Allow_NextStep THEN
				A4_Run_L	:= FALSE;
				A4_Run_P 	:= FALSE;	
				PRO_A4_[8] := PRO_A4_[8] + 10;		 
			END_IF;
		30: // CHECK ALLOW PLACE CNV NG VS
			IF ALLOW_PLACE_CNV_NG_VS THEN
				PRO_A4_[8] := PRO_A4_[8] + 10;	
			END_IF;	
		40: // XY Place NG T2
			M_CHOOSE_POS(DATA := 0, ID := 7, XYR_CONST := FALSE, Z_CONST:= TRUE); // pos 2
			IF NOT A4_Run_P THEN
				A_Comp 		:= FALSE;
				A4_Run_P 	:= TRUE;
			END_IF		
			IF MOVP_A.Error OR MOVL_A.Error THEN
				A4_Run_L	:= FALSE;
				A4_Run_P    := FALSE;	 	 
			END_IF;				
			IF A_Comp AND A4_Run_P AND A_Allow_NextStep THEN
				A4_Run_L	:= FALSE;
				A4_Run_P :=FALSE;	
				PRO_A4_[8] := PRO_A4_[8] + 10;		 
			END_IF;	
		50: // Z Place T2
			M_CHOOSE_POS(DATA := 0, ID := 7, XYR_CONST := TRUE, Z_CONST:= FALSE); // pos 2 PICK 1
			IF NOT A4_Run_P THEN
				// namnv0104
				IF NOT GVL.Pro4_.Signal_In.T_Cv_NG_out_1.Q AND NOT GVL.Pro4_.Signal_In.T_Cv_NG_out_2.Q AND NOT GVL.Pro4_.Signal_In.T_Cv_NG_out_full.Q THEN
					A_Comp	 := FALSE;
					A4_Run_P := TRUE;
				END_IF;
			END_IF	
			IF MOVP_A.Error OR MOVL_A.Error THEN
				A4_Run_L	:= FALSE;
				A4_Run_P 	:= FALSE;	 
			END_IF;			
	
			IF A_Comp AND A4_Run_P AND A_Allow_NextStep THEN
				A4_Run_L	 := FALSE;
				A4_Run_P	 := FALSE;
				A_Comp		 := FALSE;
				PRO_A4_[8] := PRO_A4_[8] + 10;		 
			END_IF;
		
		60: // OFF VACUUM
			// namnv0104
			IF NOT GVL.Pro4_.Signal_In.T_Cv_NG_out_1.Q THEN
				GVL.RB_A_.Tool_2 := FALSE;
				Project_4_Delay_A8.IN:= TRUE;
			END_IF;
			IF Project_4_Delay_A8.Q AND A_Allow_NextStep  THEN
				PRO_A4_[8] := PRO_A4_[8] + 10; 	
			END_IF;
			
		70: // BF Z Place NG T1
			M_CHOOSE_POS(DATA := 0, ID := 6, XYR_CONST := TRUE, Z_CONST:= FALSE); 
			IF NOT A4_Run_P THEN
				A_Comp	 := FALSE;
				A4_Run_P := TRUE;
			END_IF	
			IF MOVP_A.Error OR MOVL_A.Error THEN
				A4_Run_L	:= FALSE;
				A4_Run_P 	:= FALSE;	 
			END_IF;			
	
			IF A_Comp AND A4_Run_P AND A_Allow_NextStep THEN
				A4_Run_L	 := FALSE;
				A4_Run_P	 := FALSE;
				A_Comp		 := FALSE;
				PRO_A4_[8] := PRO_A4_[8] + 10;		 
			END_IF;
		80: // BF XY PPlace NG T2
			M_CHOOSE_POS(DATA := 0, ID := 6, XYR_CONST := FALSE, Z_CONST:= TRUE); // 
			IF NOT A4_Run_P THEN
				A_Comp 		:= FALSE;
				A4_Run_P 	:= TRUE;
			END_IF		
			IF MOVP_A.Error OR MOVL_A.Error THEN
				A4_Run_L	:= FALSE;
				A4_Run_P    := FALSE;	 	 
			END_IF;				
			IF A_Comp AND A4_Run_P AND A_Allow_NextStep THEN
				A4_Run_L	:= FALSE;
				A4_Run_P    := FALSE;	
				PRO_A4_[8] := PRO_A4_[8] + 10;		 
			END_IF
		
		90: // Done
			GVL.Pro4_.Process.DATA_TOOL_A2_OUT := 0;
			Project_4_Delay_A8.IN := FALSE;	
			Place_NG_TS_A4_T2_Finish    := TRUE;
			
			
	END_CASE
ELSE
	PRO_A4_[8] := 0;
END_IF
END_ACTION

ACTION B0_wait_4:
// về wait robot A (teaching Point 1)
IF Wait_B4_Run THEN
	CASE PRO_B4_[0] OF
		0: // RESET
				B4_Run_L	 := FALSE;
				B4_Run_P	 := FALSE;
				B_Comp		 := FALSE;			
				PRO_B4_[0] := PRO_B4_[0] + 10;
		10: // Z WAIT
			M_CHOOSE_POS(DATA := 1, ID := 0, XYR_CONST := TRUE, Z_CONST:= FALSE);
			IF NOT B4_Run_P THEN
				B_Comp := FALSE;
				B4_Run_P := TRUE;
			END_IF		
			IF MOVP_B.Error OR MOVL_B.Error THEN
				B4_Run_L	:= FALSE;
				B4_Run_P 	:= FALSE;	 
			END_IF;				
			IF B_Comp AND ( B4_Run_P OR B4_Run_L) AND B_Allow_NextStep THEN
				B4_Run_L	 := FALSE;
				B4_Run_P	 := FALSE;
				B_Comp		 := FALSE;
				PRO_B4_[0] := PRO_B4_[0] + 10;		 
			END_IF;
	
		20: // WAIT XY
			M_CHOOSE_POS(DATA := 1, ID := 0, XYR_CONST := FALSE, Z_CONST:= TRUE);
			IF NOT B4_Run_P THEN
				B_Comp := FALSE;
				B4_Run_P := TRUE;
			END_IF		
			IF MOVP_B.Error OR MOVL_B.Error THEN
				B4_Run_L	:= FALSE;
				B4_Run_P :=FALSE;	 	 
			END_IF;				
			IF B_Comp AND B4_Run_P AND B_Allow_NextStep THEN
				B4_Run_L	:= FALSE;
				B4_Run_P :=FALSE;	
				PRO_B4_[0] := PRO_B4_[0] + 10;			 
			END_IF;
	
		30:
			Wait_B4_Finish := TRUE;
		
	END_CASE
ELSE
	PRO_B4_[0] := 0;
END_IF
END_ACTION

ACTION B1_Pick_T1_4:
Project_4_Delay_B1(PT := TO_TIME(GVL.Pro4_.ST_B.TDelay_pick_T1)*100, Q =>, ET =>);
IF Pick_B4_Run THEN
	CASE PRO_B4_[1] OF
		0: // RESET
				B4_Run_L	 := FALSE;
				B4_Run_P	 := FALSE;
				B_Comp		 := FALSE;		
				Project_4_Delay_B1.IN := FALSE;	
				PRO_B4_[1] := PRO_B4_[1] + 10;
		10: // XY PICK
			M_CHOOSE_POS(DATA := 1, ID := 1, XYR_CONST := FALSE, Z_CONST:= TRUE); // 
			IF NOT B4_Run_P THEN
				B_Comp := FALSE;
				B4_Run_P := TRUE;
			END_IF		
			IF MOVP_B.Error OR MOVL_B.Error THEN
				B4_Run_L	:= FALSE;
				B4_Run_P 	:= FALSE;	 
			END_IF;				
			IF B_Comp AND B4_Run_P AND B_Allow_NextStep THEN
				B4_Run_L	 := FALSE;
				B4_Run_P	 := FALSE;
				B_Comp		 := FALSE;
				PRO_B4_[1] := PRO_B4_[1] + 10;		 
			END_IF;
	
		20: // PICK Z
			M_CHOOSE_POS(DATA := 1, ID := 1, XYR_CONST := TRUE, Z_CONST:= FALSE); // pos 1
			IF NOT B4_Run_P THEN
				B_Comp := FALSE;
				B4_Run_P := TRUE;
			END_IF		
			IF MOVP_B.Error OR MOVL_B.Error THEN
				B4_Run_L	:= FALSE;
				B4_Run_P :=FALSE;	 	 
			END_IF;				
			IF B_Comp AND B4_Run_P AND B_Allow_NextStep THEN
				B4_Run_L	:= FALSE;
				B4_Run_P :=FALSE;	
				PRO_B4_[1] := PRO_B4_[1] + 10;		 
			END_IF;
	
		30: // ON VACUUM
			IF (NOT GVL.Pro4_.ST_MC.Mode_Dry) THEN
				GVL.RB_B_.Tool_1 := TRUE;
			END_IF;
			Project_4_Delay_B1.IN := TRUE;
			IF Project_4_Delay_B1.Q AND B_Allow_NextStep AND (GVL.RB_Signal_In.SS_RBB_Tool_1.Q OR GVL.Pro4_.ST_MC.Mode_Skip_ss_T1_b) THEN
				PRO_B4_[1] := PRO_B4_[1] + 10; 	
			END_IF;
			
		40: // Z WAIT
			
			IF (GVL.Pro4_.ST_MC.Mode_Skip_VS_Align) THEN
				GVL.Pro4_.Process.DATA_TOOL_B1_IN := 3; // cho Doc bar code luon
			ELSE
				GVL.Pro4_.Process.DATA_TOOL_B1_IN := 1; // cho trigger Vision
			END_IF;
			Project_4_Delay_B1.IN := FALSE;
			M_CHOOSE_POS(DATA := 1, ID := 0, XYR_CONST := TRUE, Z_CONST:= FALSE); // pos wait
			IF NOT B4_Run_P THEN
				B_Comp := FALSE;
				B4_Run_P := TRUE;
			END_IF		
			IF MOVP_B.Error OR MOVL_B.Error THEN
				B4_Run_L	:= FALSE;
				B4_Run_P 	:= FALSE;	 
			END_IF;				
			IF B_Comp AND B4_Run_P AND B_Allow_NextStep THEN
				B4_Run_L	 := FALSE;
				B4_Run_P	 := FALSE;
				B_Comp		 := FALSE;
				PRO_B4_[1] := PRO_B4_[1] + 10;		 
			END_IF;		
		50:
			Pick_B4_Finish := TRUE;
			
			
	END_CASE
ELSE
	PRO_B4_[1] := 0;
END_IF
END_ACTION

ACTION B2_PLace_T1_4:
Project_4_Delay_B2( PT := TO_TIME(GVL.Pro4_.ST_B.TDelay_Place_T1)*100);
IF Place_B4_Run THEN
	CASE PRO_B4_[2] OF
		0: // RESET
				B4_Run_L	 := FALSE;
				B4_Run_P	 := FALSE;
				B_Comp		 := FALSE;	
				Project_4_Delay_B2.IN := FALSE;		
				PRO_B4_[2] := PRO_B4_[2] + 10;
		10: // Befor Place Z
			M_CHOOSE_POS(DATA := 1, ID := 2, XYR_CONST := TRUE, Z_CONST:= FALSE); // pos 2
			IF NOT B4_Run_P THEN
				B_Comp := FALSE;
				B4_Run_P := TRUE;
			END_IF		
			IF MOVP_B.Error OR MOVL_B.Error THEN
				B4_Run_L	:= FALSE;
				B4_Run_P 	:= FALSE;	 
			END_IF;				
			IF B_Comp AND B4_Run_P AND B_Allow_NextStep THEN
				B4_Run_L	 := FALSE;
				B4_Run_P	 := FALSE;
				B_Comp		 := FALSE;
				PRO_B4_[2] := PRO_B4_[2] + 10;		 
			END_IF;
	
		20: // Befor Place Xy
			M_CHOOSE_POS(DATA := 1, ID := 2, XYR_CONST := FALSE, Z_CONST:= TRUE); // pos 2
// 			IF (NOT GVL.Pro4_.ST_MC.Mode_Skip_VS_Align) THEN
// 				M_CHOOSE_POS(DATA := 1, ID := 2, XYR_CONST := FALSE, Z_CONST:= TRUE); // pos 2
// 			ELSE
// 				M_CHOOSE_POS_VS(DATA := 1, ID := 2, XYR_CONST := FALSE, Z_CONST:= TRUE); // pos 2
// 			END_IF;
			IF NOT B4_Run_P THEN
				B_Comp := FALSE;
				B4_Run_P := TRUE;
			END_IF		
			IF MOVP_B.Error OR MOVL_B.Error THEN
				B4_Run_L	:= FALSE;
				B4_Run_P :=FALSE;	 	 
			END_IF;				
			IF B_Comp AND B4_Run_P AND B_Allow_NextStep THEN
				B4_Run_L	:= FALSE;
				B4_Run_P :=FALSE;	
				PRO_B4_[2] := PRO_B4_[2] + 10;		 
			END_IF;
		30:  // kiểm tra MC 1 cho phép đặt hàng
			IF GVL.Pro4_.Process.DATA_MC_TS = 2 AND GVL.Pro4_.Signal_In.T_Ts_Press_Up.Q THEN
				change_fac_vel_max_B := TRUE; //namnv0204
				PRO_B4_[2] := PRO_B4_[2] + 10; 	
			END_IF
		40: // xy place
			IF (GVL.Pro4_.ST_MC.Mode_Skip_VS_Align) THEN
				M_CHOOSE_POS(DATA := 1, ID := 3, XYR_CONST := FALSE, Z_CONST:= TRUE); // pos 3
			ELSE
				M_CHOOSE_POS_VS(DATA := 1, ID := 3, XYR_CONST := FALSE, Z_CONST:= TRUE); // pos 3
			END_IF;
// 			IF NOT B4_Run_P THEN
			IF NOT B4_Run_P AND (GVL.Fac_Vel_Set_B = GVL.Pro4_.Auto.Fac_Vel_Max_B) THEN
				B_Comp := FALSE;
				IF NOT NextStep_Test_1 THEN
					B4_Run_P := TRUE;
				END_IF;
			END_IF		
			IF MOVP_B.Error OR MOVL_B.Error THEN
				B4_Run_L	:= FALSE;
				B4_Run_P :=FALSE;	 	 
			END_IF;				
			IF B_Comp AND B4_Run_P AND B_Allow_NextStep THEN
				B4_Run_L	:= FALSE;
				B4_Run_P :=FALSE;	
				PRO_B4_[2] := PRO_B4_[2] + 15;		 
			END_IF;
		50: // z place BF 10mm
			//M_CHOOSE_POS(DATA := 1, ID := 3, XYR_CONST := TRUE, Z_CONST:= FALSE); // pos 3
			M_CHOOSE_POS_Z_BF(DATA := 1, ID := 3, XYR_CONST := TRUE, Z_CONST:= FALSE);
			IF NOT B4_Run_P THEN
				B_Comp := FALSE;
				B4_Run_P := TRUE;
			END_IF		
			IF MOVP_B.Error OR MOVL_B.Error THEN
				B4_Run_L	:= FALSE;
				B4_Run_P :=FALSE;	 	 
			END_IF;				
			IF B_Comp AND B4_Run_P AND B_Allow_NextStep THEN
				B4_Run_L	:= FALSE;
				B4_Run_P :=FALSE;	
				PRO_B4_[2] := PRO_B4_[2] + 5;		 
			END_IF;			
		55: // z place T1
			//change_fac_vel_B := TRUE;
			M_CHOOSE_POS(DATA := 1, ID := 3, XYR_CONST := TRUE, Z_CONST:= FALSE); // pos 3
			IF NOT B4_Run_P THEN
				B_Comp := FALSE;
				B4_Run_P := TRUE;
			END_IF		
			IF MOVP_B.Error OR MOVL_B.Error THEN
				B4_Run_L	:= FALSE;
				B4_Run_P :=FALSE;	 	 
			END_IF;				
			IF B_Comp AND B4_Run_P AND B_Allow_NextStep THEN
				B4_Run_L	:= FALSE;
				B4_Run_P :=FALSE;	
				PRO_B4_[2] := PRO_B4_[2] + 5;		 
				change_fac_vel_B := FALSE;
			END_IF;		
		60: // OFF VACUUM
			GVL.RB_B_.Tool_1 := FALSE;
			Project_4_Delay_B2.IN:= TRUE ;
			IF Project_4_Delay_B2.Q AND B_Allow_NextStep  THEN
				PRO_B4_[2] := PRO_B4_[2] + 10; 	
			END_IF;	
		70: // Z befor
			
			Project_4_Delay_B2.IN := FALSE;
			M_CHOOSE_POS(DATA := 1, ID := 2, XYR_CONST := TRUE, Z_CONST:= FALSE); // pos 2
			IF NOT B4_Run_P THEN
				B_Comp := FALSE;
				B4_Run_P := TRUE;
			END_IF		
			IF MOVP_B.Error OR MOVL_B.Error THEN
				B4_Run_L	:= FALSE;
				B4_Run_P 	:= FALSE;	 
			END_IF;				
			IF B_Comp AND B4_Run_P AND B_Allow_NextStep THEN
				B4_Run_L	 := FALSE;
				B4_Run_P	 := FALSE;
				B_Comp		 := FALSE;
				PRO_B4_[2] := PRO_B4_[2] + 10;		 
			END_IF;	
		80: // xy befor place
			M_CHOOSE_POS(DATA := 1, ID := 2, XYR_CONST := FALSE, Z_CONST:= TRUE); // pos 2
			IF NOT B4_Run_P THEN
				B_Comp := FALSE;
				B4_Run_P := TRUE;
			END_IF		
			IF MOVP_B.Error OR MOVL_B.Error THEN
				B4_Run_L	:= FALSE;
				B4_Run_P :=FALSE;	 	 
			END_IF;				
			IF B_Comp AND B4_Run_P AND B_Allow_NextStep THEN
				B4_Run_L	:= FALSE;
				B4_Run_P :=FALSE;	
				PRO_B4_[2] := PRO_B4_[2] + 10;		 
				change_fac_vel_max_B := FALSE; //namnv0204
			END_IF;		
		90: // Z wait
			change_fac_vel_max_B := FALSE; //namnv0204
			GVL.Pro4_.Process.DATA_TOOL_B1_IN := 0;
			M_CHOOSE_POS(DATA := 1, ID := 0, XYR_CONST := TRUE, Z_CONST:= FALSE);
			IF NOT B4_Run_P THEN
				B_Comp := FALSE;
				B4_Run_P := TRUE;
			END_IF		
			IF MOVP_B.Error OR MOVL_B.Error THEN
				B4_Run_L	:= FALSE;
				B4_Run_P 	:= FALSE;	 
			END_IF;				
			IF B_Comp AND B4_Run_P AND B_Allow_NextStep THEN
				B4_Run_L	 := FALSE;
				B4_Run_P	 := FALSE;
				B_Comp		 := FALSE;
				PRO_B4_[2] := PRO_B4_[2] + 10;	
				Monitor_Production.Pulse_In := FALSE;
				Monitor_Production.Pulse_Out := TRUE;	 
			END_IF;		
		100: // finish
			Place_B4_Finish := TRUE;
			Monitor_Production.Pulse_In := TRUE;
			Monitor_Production.Pulse_Out := FALSE;
	
	END_CASE
ELSE
	PRO_B4_[2] := 0;
END_IF
END_ACTION

ACTION B3_Barcode_4:
//Project_4_Delay_B3(PT := TO_TIME(GVL.Pro4_.ST_MC.Delay_Trigger_Barcode_Ts)*100);
T_Wait_Trigger_Bar_TS( PT := TO_TIME(GVL.Pro4_.ST_MC.Delay_Trigger_Barcode_Ts)*100);
IF Barcode_B4_Run THEN
	CASE PRO_B4_[3] OF
		0: // RESET
				B4_Run_L	 := FALSE;
				B4_Run_P	 := FALSE;
				B_Comp		 := FALSE;	
				//Project_4_Delay_B3.in := FALSE;		
				count_Ts := 0;  // namnv 
				PRO_B4_[3] := PRO_B4_[3] + 10;
		10: // XY barcode
			IF (GVL.Pro4_.ST_MC.Mode_Skip_VS_Align) THEN
				M_CHOOSE_POS(DATA := 1, ID := 4, XYR_CONST := FALSE, Z_CONST:= TRUE); // pos 4 barcode
			ELSE
				M_CHOOSE_POS_VS(DATA := 1, ID := 4, XYR_CONST := FALSE, Z_CONST:= TRUE);
			END_IF;
			IF NOT B4_Run_P THEN
				B_Comp := FALSE;
				IF NOT NextStep_Test THEN
					B4_Run_P := TRUE;
				END_IF;
			END_IF		
			IF MOVP_B.Error OR MOVL_B.Error THEN
				B4_Run_L	:= FALSE;
				B4_Run_P 	:= FALSE;	 
			END_IF;				
			IF B_Comp AND B4_Run_P AND A_Allow_NextStep THEN
				B4_Run_L	 := FALSE;
				B4_Run_P	 := FALSE;
				B_Comp		 := FALSE;
				PRO_B4_[3] := PRO_B4_[3] + 10;		 
			END_IF;
	
		20: // Barcode Z
			
			M_CHOOSE_POS(DATA := 1, ID := 4, XYR_CONST := TRUE, Z_CONST:= FALSE); // pos 4 barcode
			IF NOT B4_Run_P THEN
				B_Comp := FALSE;
				B4_Run_P := TRUE;
			END_IF		
			IF MOVP_B.Error OR MOVL_B.Error THEN
				B4_Run_L	:= FALSE;
				B4_Run_P :=FALSE;	 	 
			END_IF;				
			IF B_Comp AND B4_Run_P AND A_Allow_NextStep THEN
				B4_Run_L	:= FALSE;
				B4_Run_P :=FALSE;	
				PRO_B4_[3] := PRO_B4_[3] + 10;		 
			END_IF;
	
		30: // Trigger Barcode
			// Ontrigger
			CASE D_Barcode_Ts OF
				0:
					IF GVL.Pro4_.ST_MC.Mode_Skip_Barcode_ts THEN
						D_Barcode_Ts := 30;
					ELSE
							GVL.Pro4_.Auto.Trigger_Barcode_Ts_On_Off := 1;
							//Project_4_Delay_B3.IN := TRUE;
						//IF GVL.Pro4_.Auto.Trigger_Barcode_Ts_On_Off = 1 AND Project_4_Delay_B3.q THEN	
						IF GVL.Pro4_.Auto.Trigger_Barcode_Ts_On_Off = 1 THEN
							D_Barcode_Ts := D_Barcode_Ts +10;
						END_IF						
					END_IF

				10:
					//Project_4_Delay_B3.IN := FALSE;
					GVL.Pro4_.Auto.Trigger_Barcode_Ts_On_Off := 0;
					IF GVL.Pro4_.Auto.Trigger_Barcode_Ts_On_Off = 0 THEN
						count_Ts := count_Ts +1;
						D_Barcode_Ts := D_Barcode_Ts +10;
						T_Wait_Trigger_Bar_TS.IN := TRUE;
					END_IF
				20:
					IF GVL.Pro4_.Signal_In.T_Ts_Result_Scanner.Q OR  GVL.X[31] THEN
						D_Barcode_Ts := D_Barcode_Ts +10;
						T_Wait_Trigger_Bar_TS.IN := FALSE;
					ELSIF NOT GVL.Pro4_.Signal_In.T_Ts_Result_Scanner.Q AND NOT GVL.X[31]  AND count_Ts <= 5 AND T_Wait_Trigger_Bar_TS.Q THEN
						D_Barcode_Ts := 0;
						T_Wait_Trigger_Bar_TS.IN := FALSE;
					END_IF
				30:
					// ok	
			END_CASE;
			IF count_Ts > 5 AND (GVL.X[8] OR gvl.Pro4_.Process.Re_Trigger_Barcode_Ts) THEN
				count_Ts := 0;
			END_IF
			IF count_Ts > 5 AND D_Barcode_Ts = 20 AND NOT GVL.Pro4_.Auto.Alarm_Not_barcode  THEN
				GVL.Pro4_.Auto.Alarm_Not_barcode := TRUE;
			ELSIF GVL.Pro4_.Auto.Alarm_Not_barcode AND GVL.Pro4_.Auto.comfirm_Reduct_Pro THEN
				count_Ts:=0;
				PRO_B4_[3] := 50; 	
			END_IF
			

			IF D_Barcode_Ts = 30 AND A_Allow_NextStep  THEN
				count_Ts:=0;
				PRO_B4_[3] := PRO_B4_[3] + 10; 	
			END_IF;
			
		40: // Z WAIT
			
			D_Barcode_Ts := 0;
			//Project_4_Delay_B3.IN := FALSE;
			M_CHOOSE_POS(DATA := 1, ID := 0, XYR_CONST := TRUE, Z_CONST:= FALSE); // pos wait
			IF NOT B4_Run_P THEN
				B_Comp := FALSE;
				B4_Run_P := TRUE;
			END_IF		
			IF MOVP_B.Error OR MOVL_B.Error THEN
				B4_Run_L	:= FALSE;
				B4_Run_P 	:= FALSE;	 
			END_IF;				
			IF B_Comp AND B4_Run_P AND A_Allow_NextStep THEN
				B4_Run_L	 := FALSE;
				B4_Run_P	 := FALSE;
				B_Comp		 := FALSE;
				PRO_B4_[3] := PRO_B4_[3] + 10;		 
			END_IF;		
		50:
			IF GVL.Pro4_.Auto.comfirm_Reduct_Pro THEN
				GVL.Pro4_.Process.DATA_TOOL_B1_IN := 0; // trigger barcode OK
			ELSE 
				GVL.Pro4_.Process.DATA_TOOL_B1_IN := 2; // trigger barcode OK
			END_IF
			GVL.Pro4_.Auto.Alarm_Not_barcode := FALSE;
			Barcode_B4_Finish := TRUE;
			
			
	END_CASE
ELSE
	PRO_B4_[3] := 0;
END_IF
END_ACTION

ACTION B_Trigger_4:
Trigger_Auto_Done(CLK:= GVL.Pro4_.Auto.Result_Trigger_Vs_Align_Done);
Project_4_Delay_B4(PT := TO_TIME(GVL.Pro4_.ST_MC.Delay_Trigger_Vision_Align)*100);
IF Trigger_B4_Run THEN
	CASE PRO_B4_[4] OF
		0: // RESET
				B4_Run_L	 := FALSE;
				B4_Run_P	 := FALSE;
				B_Comp		 := FALSE;	
				//Project_4_Delay_B4.in := FALSE;		
				count_Vs_Align := 0;  // namnv 
				IF NOT GVL.Pro4_.Auto.Result_Trigger_Vs_Align_Done THEN
					PRO_B4_[4] := PRO_B4_[4] + 10;
				END_IF;
		10: // XY Vision
			M_CHOOSE_POS(DATA := 1, ID := 5, XYR_CONST := FALSE, Z_CONST:= TRUE); // pos 5 Vision Trigger
			IF NOT B4_Run_P THEN
				B_Comp := FALSE;
				B4_Run_P := TRUE;
			END_IF		
			IF MOVP_B.Error OR MOVL_B.Error THEN
				B4_Run_L	:= FALSE;
				B4_Run_P 	:= FALSE;	 
			END_IF;				
			IF B_Comp AND B4_Run_P AND A_Allow_NextStep THEN
				B4_Run_L	 := FALSE;
				B4_Run_P	 := FALSE;
				B_Comp		 := FALSE;
				PRO_B4_[4] := PRO_B4_[4] + 10;		 
			END_IF;
	
		20: // Vision Z
			
			M_CHOOSE_POS(DATA := 1, ID := 5, XYR_CONST := TRUE, Z_CONST:= FALSE); // pos 5 vision
			IF NOT B4_Run_P THEN
				B_Comp := FALSE;
				B4_Run_P := TRUE;
			END_IF		
			IF MOVP_B.Error OR MOVL_B.Error THEN
				B4_Run_L	:= FALSE;
				B4_Run_P :=FALSE;	 	 
			END_IF;				
			IF B_Comp AND B4_Run_P AND A_Allow_NextStep THEN
				B4_Run_L	:= FALSE;
				B4_Run_P :=FALSE;	
				PRO_B4_[4] := PRO_B4_[4] + 10;		 
			END_IF;
	
		30: // Trigger Vision
			// Ontrigger
			CASE D_Vision_Align_Ts OF
				0:
					IF GVL.Pro4_.ST_MC.Mode_Skip_VS_Align THEN
						D_Vision_Align_Ts := 30;
					ELSE
							GVL.Pro4_.Auto.Trigger_Vs_Align_On_Off := 1;
							Project_4_Delay_B4.IN := TRUE;
						IF GVL.Pro4_.Auto.Trigger_Vs_Align_On_Off = 1 AND Project_4_Delay_B4.q THEN
							D_Vision_Align_Ts := D_Vision_Align_Ts +10;
						END_IF						
					END_IF

				10:
					Project_4_Delay_B4.IN := FALSE;
					D_Vision_Align_Ts := D_Vision_Align_Ts +10;
// 					IF GVL.Pro4_.Auto.Trigger_Vs_Align_On_Off = 0 THEN
// 						count_Vs_Align := count_Vs_Align +1;
// 						D_Vision_Align_Ts := D_Vision_Align_Ts +10;
// 					END_IF
				20:
					IF GVL.Pro4_.Auto.Result_Trigger_Vs_Align_Done THEN
						D_Vision_Align_Ts := D_Vision_Align_Ts +10;
						GVL.Pro4_.Auto.Trigger_Vs_Align_On_Off := 0;
					ELSIF NOT GVL.Pro4_.Auto.Result_Trigger_Vs_Align_Done AND count_Vs_Align <= 5 THEN
						D_Vision_Align_Ts := 0;
						count_Vs_Align := count_Vs_Align +1;
						GVL.Pro4_.Auto.Trigger_Vs_Align_On_Off := 0;
					END_IF
				30:
					// ok	
			END_CASE;
			IF count_Vs_Align > 5 AND (GVL.X[8] OR gvl.Pro4_.Process.Re_Trigger_VS_Align) THEN
				count_Vs_Align := 0;
			END_IF
			IF count_Vs_Align > 5 AND D_Vision_Align_Ts = 20 AND NOT GVL.Pro4_.Auto.Alarm_VS_Align  THEN
				GVL.Pro4_.Auto.Alarm_VS_Align := TRUE;
				GVL.Pro4_.Auto.Trigger_Vs_Align_On_Off := 0;
			ELSIF GVL.Pro4_.Auto.Alarm_VS_Align AND GVL.Pro4_.Auto.comfirm_Reduct_Pro_NG_Vs_Align THEN
				count_Vs_Align:=0;
				PRO_B4_[4] := 50; 	
			END_IF
			

			IF D_Vision_Align_Ts = 30 AND A_Allow_NextStep  THEN
				count_Vs_Align:=0;
				PRO_B4_[4] := PRO_B4_[4] + 10; 	
			END_IF;
			
		40: // Z WAIT
			
			D_Vision_Align_Ts := 0;
			Project_4_Delay_B4.IN := FALSE;
			M_CHOOSE_POS(DATA := 1, ID := 0, XYR_CONST := TRUE, Z_CONST:= FALSE); // pos wait
			IF NOT B4_Run_P THEN
				B_Comp := FALSE;
				B4_Run_P := TRUE;
			END_IF		
			IF MOVP_B.Error OR MOVL_B.Error THEN
				B4_Run_L	:= FALSE;
				B4_Run_P 	:= FALSE;	 
			END_IF;				
			IF B_Comp AND B4_Run_P AND A_Allow_NextStep THEN
				B4_Run_L	 := FALSE;
				B4_Run_P	 := FALSE;
				B_Comp		 := FALSE;
				PRO_B4_[4] := PRO_B4_[4] + 10;		 
			END_IF;		
		50:
			IF GVL.Pro4_.Auto.comfirm_Reduct_Pro_NG_Vs_Align THEN
				GVL.Pro4_.Process.DATA_TOOL_B1_IN := 0; // trigger Vision NG, bo hang ra
			ELSE 
				GVL.Pro4_.Process.DATA_TOOL_B1_IN := 3; // trigger Vision OK
			END_IF
			GVL.Pro4_.Auto.Alarm_VS_Align := FALSE;
			Trigger_B4_Finish := TRUE;
			
			
	END_CASE
ELSE
	PRO_B4_[4] := 0;
END_IF


// // ALLOW_PICK_CNV_4 := GVL.X[27];
// IF Trigger_Cmd THEN
// 	Trigger_Busy := TRUE;
// 	GVL_2.Process3.Trigger := TRUE;
// 	
// 	IF GVL.MODBUS[100].5 THEN 
// 		GVL_2.Process3.Shape_T1 := 1;
// 	ELSIF GVL.MODBUS[100].6 THEN
// 		GVL_2.Process3.Shape_T1 := 2;
// 	ELSIF GVL.MODBUS[100].7 THEN
// 		GVL_2.Process3.Shape_T1 := 3;	
// 	ELSIF GVL.MODBUS[100].8 THEN
// 		GVL_2.Process3.Shape_T1 := 4;
// 	ELSE
// 		GVL_2.Process3.Shape_T1 := 0;
// 	END_IF;
// 	
// 	IF GVL.MODBUS[100].12 THEN 
// 		GVL_2.Process3.Shape_T2 := 1;
// 	ELSIF GVL.MODBUS[100].13 THEN
// 		GVL_2.Process3.Shape_T2 := 2;
// 	ELSIF GVL.MODBUS[100].14 THEN
// 		GVL_2.Process3.Shape_T2 := 3;	
// 	ELSIF GVL.MODBUS[100].15 THEN
// 		GVL_2.Process3.Shape_T2 := 4;
// 	ELSE
// 		GVL_2.Process3.Shape_T2 := 0;
// 	END_IF;
// // 	GVL_2.pro3_B_get.Pos_Target_T1.X :=  GVL.Cam_T1.POS_X_RESULT + GVL_2.pro3_B_get.Pos_vision_T1_Offset.X;
// // 	GVL_2.pro3_B_get.Pos_Target_T1.Y :=  GVL.Cam_T1.POS_Y_RESULT + GVL_2.pro3_B_get.Pos_vision_T1_Offset.Y;
// // 	GVL_2.pro3_B_get.Pos_Target_T1.Z :=  GVL_2.pro3_B_get.Pos_vision_T1.Z + GVL_2.pro3_B_get.Pos_vision_T1_Offset.Z;					 
// // 	GVL_2.pro3_B_get.Pos_Target_T1.A :=  GVL_2.pro3_B_get.Pos_vision_T1.A + GVL_2.pro3_B_get.Pos_vision_T1_Offset.A;	
// // 	
// // 	GVL_2.pro3_B_get.Pos_Target_T2.X :=  GVL.Cam_T2.POS_X_RESULT + GVL_2.pro3_B_get.Pos_vision_T2_Offset.X;
// // 	GVL_2.pro3_B_get.Pos_Target_T2.Y :=  GVL.Cam_T2.POS_Y_RESULT + GVL_2.pro3_B_get.Pos_vision_T2_Offset.Y;
// // 	GVL_2.pro3_B_get.Pos_Target_T2.Z :=  GVL_2.pro3_B_get.Pos_vision_T2.Z + GVL_2.pro3_B_get.Pos_vision_T2_Offset.Z;				 
// // 	GVL_2.pro3_B_get.Pos_Target_T2.A :=  GVL_2.pro3_B_get.Pos_vision_T2.A + GVL_2.pro3_B_get.Pos_vision_T2_Offset.A;
// ELSE
// 	GVL_2.Process3.Trigger := FALSE;
// 	Trigger_Done := FALSE;
// END_IF;

// 	GVL_2.pro3_B_get.Pos_Target_T1.X :=  GVL.Cam_T1.POS_X_RESULT + GVL_2.pro3_B_get.Pos_vision_T1_Offset.X;
// 	GVL_2.pro3_B_get.Pos_Target_T1.Y :=  GVL.Cam_T1.POS_Y_RESULT + GVL_2.pro3_B_get.Pos_vision_T1_Offset.Y;
// 	GVL_2.pro3_B_get.Pos_Target_T1.Z :=  GVL_2.pro3_B_get.Pos_vision_T1.Z + GVL_2.pro3_B_get.Pos_vision_T1_Offset.Z;					 
// 	GVL_2.pro3_B_get.Pos_Target_T1.A :=  GVL_2.pro3_B_get.Pos_vision_T1.A + GVL_2.pro3_B_get.Pos_vision_T1_Offset.A;	
// 	
// 	GVL_2.pro3_B_get.Pos_Target_T2.X :=  GVL.Cam_T2.POS_X_RESULT + GVL_2.pro3_B_get.Pos_vision_T2_Offset.X;
// 	GVL_2.pro3_B_get.Pos_Target_T2.Y :=  GVL.Cam_T2.POS_Y_RESULT + GVL_2.pro3_B_get.Pos_vision_T2_Offset.Y;
// 	GVL_2.pro3_B_get.Pos_Target_T2.Z :=  GVL_2.pro3_B_get.Pos_vision_T2.Z + GVL_2.pro3_B_get.Pos_vision_T2_Offset.Z;				 
// 	GVL_2.pro3_B_get.Pos_Target_T2.A :=  GVL_2.pro3_B_get.Pos_vision_T2.A + GVL_2.pro3_B_get.Pos_vision_T2_Offset.A;
END_ACTION

ACTION CNV_NG:
T_distance_NG(PT:= T#200MS);

IF GVL.Pro4_.Signal_In.T_Cv_NG_out_full.Q THEN
	GVL.Pro4_.Auto.Cv_NG_On_Off := FALSE;
	//GVL.Pro4_.Auto.NG_CV_Full_Pro := TRUE;
	RETURN;
ELSE
	//GVL.Pro4_.Auto.NG_CV_Full_Pro := FALSE;
	IF GVL.Pro4_.Signal_In.T_Cv_NG_out_1.Q THEN
		GVL.Pro4_.Auto.Cv_NG_On_Off := TRUE;
		T_distance_NG.IN :=TRUE;
	END_IF;
// 	ELSIF (GVL.Pro4_.Signal_In.T_Cv_NG_out_2.Q AND NOT GVL.Pro4_.Signal_In.T_Cv_NG_out_1.Q ) OR T_distance_NG.Q THEN
//	ELSIF (NOT GVL.Pro4_.Signal_In.T_Cv_NG_out_1.Q AND T_distance_NG.Q) THEN
//  	IF ( GVL.Pro4_.Signal_In.T_Cv_NG_out_2.Q ) THEN
// 		T_distance_NG.IN :=TRUE;		
// 	END_IF
	IF T_distance_NG.Q AND NOT GVL.Pro4_.Signal_In.T_Cv_NG_out_2.Q THEN
		T_distance_NG.IN := FALSE;
		GVL.Pro4_.Auto.Cv_NG_On_Off := FALSE;
	END_IF
END_IF
END_ACTION

ACTION Pro_MC1_4_:
T_MC1_4( PT := T#3S, Q =>, ET =>);
ton_centering (PT := T#1S, Q =>, ET =>);
Ton_OK_MC1_4( PT := T#10S);
Ton_Limit_Test_TS(PT := T#50S);
CASE Pro_MC1_4 OF
		0: // Check Data
			T_MC1_4.IN := FALSE;
			ton_centering.IN := FALSE;
			Ton_OK_MC1_4.IN := FALSE;
			Ton_Limit_Test_TS.IN := FALSE;
			//GVL.Pro4_.Process.DATA_MC_TS := 0;
			on_centering := 0;
			Pro_MC1_4 := 5;
			
		5:
			T_MC1_4.IN := FALSE;
			CASE GVL.Pro4_.Process.DATA_MC_TS OF
				0 : // None
					Pro_MC1_4 := 10;
				1: // Busy - checking
					Pro_MC1_4 := 20;
				2: // Allow Place
					Pro_MC1_4 := 30;
				3: // Allow Pick OK
					Pro_MC1_4 := 40;
				4: // Allow Pick NG
					Pro_MC1_4 := 50;
			END_CASE;
		10: // init - Stop - cylinder press UP
			//IF GVL.X[24] AND NOT GVL.X[25] THEN
			IF  GVL.Pro4_.Signal_In.T_Ts_Press_Up.Q  THEN
				T_MC1_4.IN := FALSE;
				GVL.Pro4_.Auto.TS_On_Off := FALSE;
				GVL.Pro4_.Process.DATA_MC_TS := 2 ; // allow place
				Pro_MC1_4 := 5;
			END_IF;
		20: // Checking
			CASE on_centering OF
				0 : 
					GVL.Pro4_.Auto.centering_ts_On_Off  := TRUE;
					on_centering := on_centering + 10;
				10: 
					ton_centering.IN := TRUE;
					IF (ton_centering.Q ) THEN
						on_centering := on_centering + 10;
						Ton_Limit_Test_TS.IN := TRUE;
					END_IF
				20:
					GVL.Pro4_.Auto.centering_ts_On_Off  := FALSE;
			END_CASE
			IF on_centering = 20 AND (GVL.Pro4_.ST_MC.Mode_Dry OR GVL.Pro4_.ST_MC.Mode_Auto_Pass_TS OR GVL.Pro4_.ST_MC.Mode_ByPass_TS) THEN
				Ton_OK_MC1_4.IN := TRUE;
				
			END_IF
			// namnv - Them dieu kien tat tin hieu start may test song
			IF  NOT GVL.Pro4_.Signal_In.T_Ts_Press_Up.Q THEN
				GVL.Pro4_.Auto.TS_On_Off := FALSE;
			END_IF
			
			//IF  T_MC1.q AND DATA_A_T1 = 0 AND GVL.X[24] AND ( GVL.X[21] OR GVL.X[22]) THEN
			IF  on_centering = 20 AND GVL.Pro4_.Signal_In.T_Ts_Press_Up.Q AND ( GVL.Pro4_.Signal_In.T_Ts_Pass.Q) AND (NOT GVL.Pro4_.ST_MC.Mode_Dry) AND (NOT GVL.Pro4_.ST_MC.Mode_ByPass_TS) THEN
				//GVL.Pro4_.Auto.centering_ts_On_Off  := TRUE;
				ton_centering.IN := FALSE;
				GVL.Pro4_.Auto.TS_On_Off := FALSE;
				GVL.Pro4_.Process.DATA_MC_TS := 3 ;
				//GVL.Pro4_.Process.DATA_MC_TS := 4 ; // namnv
				on_centering := 0;
				Pro_MC1_4 := 5;
				//namnv1104
				Monitor_Production.Pulse_In_1 := FALSE;
				Monitor_Production.Pulse_Out_1 := TRUE;
				
				
			ELSIF  on_centering = 20 AND GVL.Pro4_.Signal_In.T_Ts_Press_Up.Q  AND GVL.Pro4_.Signal_In.T_Ts_Fail.Q AND (NOT GVL.Pro4_.ST_MC.Mode_Dry) AND (NOT GVL.Pro4_.ST_MC.Mode_ByPass_TS) THEN
				//GVL.Pro4_.Auto.centering_ts_On_Off  := TRUE;
				ton_centering.IN := FALSE;
				
				GVL.Pro4_.Auto.TS_On_Off := FALSE;
				IF (GVL.Pro4_.ST_MC.Mode_Auto_Pass_TS) THEN
					IF (Ton_OK_MC1_4.Q) THEN
					GVL.Pro4_.Process.DATA_MC_TS := 3;
					END_IF;
				ELSE
					GVL.Pro4_.Process.DATA_MC_TS := 4;
				END_IF
				
				on_centering := 0;
				
				Pro_MC1_4 := 5;	
				//namnv1104
				Monitor_Production.Pulse_In_1 := FALSE;
				Monitor_Production.Pulse_Out_1 := TRUE;
			ELSIF on_centering = 20 AND GVL.Pro4_.Signal_In.T_Ts_Press_Up.Q AND (GVL.Pro4_.ST_MC.Mode_Dry OR GVL.Pro4_.ST_MC.Mode_ByPass_TS) AND Ton_OK_MC1_4.Q THEN
				ton_centering.IN := FALSE;
				GVL.Pro4_.Auto.TS_On_Off := FALSE;
				IF (Ton_OK_MC1_4.Q AND (GVL.Pro4_.ST_MC.Mode_Auto_Pass_TS OR GVL.Pro4_.ST_MC.Mode_ByPass_TS)) THEN
					GVL.Pro4_.Process.DATA_MC_TS := 3;
				ELSE
					GVL.Pro4_.Process.DATA_MC_TS := 4;
				END_IF; // namnv1504
				on_centering := 0;
				Pro_MC1_4 := 5;	
			END_IF		
			
	
		30: // Place
			IF GVL.Pro4_.Process.DATA_TOOL_B1_IN = 0 AND Place_B4_Finish THEN
				IF (NOT GVL.Pro4_.ST_MC.Mode_Dry AND NOT GVL.Pro4_.ST_MC.Mode_ByPass_TS) THEN
					GVL.Pro4_.Auto.TS_On_Off := TRUE;
				ELSE
					GVL.Pro4_.Auto.TS_On_Off := FALSE; //namnv1504
				END_IF;
				GVL.Pro4_.Auto.centering_ts_On_Off  := FALSE;
				GVL.Pro4_.Process.DATA_MC_TS := 1 ;
				Pro_MC1_4 := 5;
				//namnv1104
				Monitor_Production.Pulse_In_1 := TRUE;
				Monitor_Production.Pulse_Out_1 := FALSE;
			END_IF
		40:	// Pick OK
				GVL.Pro4_.Auto.centering_ts_On_Off  := FALSE;
			//IF GVL.Pro4_.Process.DATA_TOOL_A1_IN = 2 AND Pick_A4_T1_Finish THEN
			// namnv
			IF (GVL.Pro4_.Process.DATA_TOOL_A1_IN = 2 OR GVL.Pro4_.Process.DATA_TOOL_A1_IN = 1)  AND Pick_A4_T1_Finish THEN
				Ton_OK_MC1_4.IN := FALSE;
				Ton_Limit_Test_TS.IN := FALSE;
				GVL.Pro4_.Process.DATA_MC_TS := 0;			
				Pro_MC1_4  := 5;
			END_IF	
		50:	// Pick NG
			GVL.Pro4_.Auto.centering_ts_On_Off  := FALSE;
			IF GVL.Pro4_.Process.DATA_TOOL_A1_IN = 3 AND Pick_A4_T1_Finish THEN
				Ton_OK_MC1_4.IN := FALSE;
				Ton_Limit_Test_TS.IN := FALSE;
				GVL.Pro4_.Process.DATA_MC_TS := 0;
				Pro_MC1_4  := 5;
				
			END_IF		
	END_CASE
END_ACTION

ACTION Pro_MC2_4_:
Ton_OK_MC2_4(PT := T#5S);
T_MC2_4(PT := T#1S, Q =>, ET =>);
Ton_Limit_Test_VS(PT := T#20S);
CASE Pro_MC2_4 OF
		0: // Check Data
			T_MC2_4.IN := FALSE;
			Ton_Limit_Test_VS.IN := FALSE;
			//GVL.Pro4_.Process.DATA_MC_VS := 0;
			Ton_OK_MC2_4.IN := FALSE;
			Pro_MC2_4 := 5;
		5:
			T_MC2_4.IN := FALSE;
			CASE GVL.Pro4_.Process.DATA_MC_VS OF
				0 : // None
					Pro_MC2_4 := 10;
				1: // Busy - checking
					Pro_MC2_4 := 20;
				2: // Allow Place
					Pro_MC2_4 := 30;
				3: // Allow Pick OK
					Pro_MC2_4 := 40;
				4: // Allow Pick NG
					Pro_MC2_4 := 50;
				5: // Allow Pick NG - TS
					Pro_MC2_4 := 60;
			END_CASE;
		10: // init - Stop - cylinder press UP
			
			// IF NOT GVL.Pro4_.Signal_In.T_Vs_detect.Q THEN
			// namnv
			IF GVL.Pro4_.Signal_In.T_Vs_detect.Q THEN
				GVL.Pro4_.Auto.Vs_On_Off := FALSE;
				GVL.Pro4_.Process.DATA_MC_VS := 2 ; // allow place
				Pro_MC2_4 := 5;
			END_IF;
		20: // Checking
			Ton_OK_MC2_4.IN := TRUE;
			T_MC2_4.IN := TRUE;
			Ton_Limit_Test_VS.IN := TRUE;
			// namnv them dieu kien xac nhan Pass - Fail: Phai co tin hieu jig o ben ngoai :  AND GVL.Pro4_.Signal_In.T_Vs_detect.Q 
			IF  T_MC2_4.q AND ( GVL.Pro4_.Signal_In.T_Vs_Pass.Q) AND GVL.Pro4_.Signal_In.T_Vs_detect.Q THEN
				GVL.Pro4_.Auto.Vs_On_Off := FALSE;
				GVL.Pro4_.Process.DATA_MC_VS := 3 ;
				//GVL.Pro4_.Process.DATA_MC_VS := 4 ;  // namnv
				Pro_MC2_4  := 5;
				// namnv1104
				Monitor_Production.Pulse_In_2 := FALSE;
				Monitor_Production.Pulse_Out_2 := TRUE;
			ELSIF T_MC2_4.q AND GVL.Pro4_.Signal_In.T_Vs_Fail.Q AND GVL.Pro4_.Signal_In.T_Vs_detect.Q THEN
				GVL.Pro4_.Auto.Vs_On_Off := FALSE;
				//GVL.Pro4_.Process.DATA_MC_VS := 3 ; // namnv
				IF ((GVL.Pro4_.ST_MC.Mode_Dry OR GVL.Pro4_.ST_MC.Mode_Auto_Pass_Vs)) THEN
					IF Ton_OK_MC2_4.Q THEN
						GVL.Pro4_.Process.DATA_MC_VS := 3 ;
					END_IF;
				ELSE
					GVL.Pro4_.Process.DATA_MC_VS := 4 ;
				END_IF
				
				Pro_MC2_4  := 5;
				// namnv1104
				Monitor_Production.Pulse_In_2 := FALSE;
				Monitor_Production.Pulse_Out_2 := TRUE;
			END_IF
	
		30: // Place
			//IF GVL.Pro4_.Process.DATA_TOOL_A1_IN = 0 AND Place_OK_A4_T1_Finish  OR Place_NG_A4_T1_Finish THEN
			// namnv - bo dieu kien dat hang NG
			IF GVL.Pro4_.Process.DATA_TOOL_A1_IN = 0 AND ( Place_OK_A4_T1_Finish OR PRO_A4_[2] >= 80) THEN
				//GVL.Pro4_.Auto.Vs_On_Off := TRUE; // bat test vision
				//GVL.Pro4_.Process.DATA_MC_VS := 1 ;
				//namnv them trang thai tool
				IF (GVL.Pro4_.Process.DATA_TOOL_A1_IN_OLD = 3) THEN
					GVL.Pro4_.Process.DATA_MC_VS := 5;
				ELSIF (GVL.Pro4_.Process.DATA_TOOL_A1_IN_OLD = 2) THEN
					GVL.Pro4_.Process.DATA_MC_VS := 1 ;
					IF (GVL.Pro4_.ST_MC.Mode_Dry) THEN
						GVL.Pro4_.Auto.Vs_On_Off := FALSE; // bat test vision
					ELSE
						GVL.Pro4_.Auto.Vs_On_Off := TRUE; // bat test vision
					END_IF
					
